   DATA[1506,16] := 1.0;
   DATA[1506,17] := 1.0;
   DATA[1506,18] := 1.0;
   DATA[1506,19] := 2.0;
   DATA[1506,20] := 148.808;
   DATA[1506,21] := 153.5504;
   DATA[1506,22] := 1.711466;
   DATA[1506,23] := 789.4899;
   DATA[1506,24] := 2.0;
   DATA[1506,25] := 2.0;
   DATA[1506,26] := 7.876378;
   DATA[1506,27] := 142.707;
   DATA[1506,28] := 263.1377;
   DATA[1506,29] := 12.11228;
   DATA[1506,30] := 1.723148;
   DATA[1506,31] := 1.297041;
   DATA[1506,32] := 0.7352687;
   DATA[1506,33] := 0.3107325;
   DATA[1506,34] := 2.0;
   DATA[1506,35] := 249.984;
   DATA[1506,36] := 1.665972;
   DATA[1506,37] := 188.7657;
   DATA[1506,38] := 0.000128152;
   DATA[1506,39] := 1.0;
   DATA[1507,1] := 815.2798;
   DATA[1507,2] := 1.0;
   DATA[1507,3] := 1.0;
   DATA[1507,4] := 262.5609;
   DATA[1507,5] := 8.464369;
   DATA[1507,6] := 318.9438;
   DATA[1507,8] := 1.0;
   DATA[1507,9] := 1.0;
   DATA[1507,10] := 1.0;
   DATA[1507,11] := 19.74198;
   DATA[1507,12] := 2.210294;
   DATA[1507,13] := 939.5027;
   DATA[1507,14] := 1.0;
   DATA[1507,15] := 2.0;
   DATA[1507,16] := 1.0;
   DATA[1507,17] := 1.0;
   DATA[1507,18] := 1.0;
   DATA[1507,19] := 2.0;
   DATA[1507,20] := 148.808;
   DATA[1507,21] := 153.5504;
   DATA[1507,22] := 1.711466;
   DATA[1507,23] := 789.5283;
   DATA[1507,24] := 2.0;
   DATA[1507,25] := 2.0;
   DATA[1507,26] := 7.876378;
   DATA[1507,27] := 142.707;
   DATA[1507,28] := 263.0415;
   DATA[1507,29] := 12.11228;
   DATA[1507,30] := 1.723148;
   DATA[1507,31] := 1.290509;
   DATA[1507,32] := 0.7352687;
   DATA[1507,33] := 0.3107325;
   DATA[1507,34] := 2.0;
   DATA[1507,35] := 249.9039;
   DATA[1507,36] := 1.665972;
   DATA[1507,37] := 188.7657;
   DATA[1507,38] := 0.000128152;
   DATA[1507,39] := 1.0;
   DATA[1508,1] := 815.2013;
   DATA[1508,2] := 1.0;
   DATA[1508,3] := 1.0;
   DATA[1508,4] := 262.5609;
   DATA[1508,5] := 8.464369;
   DATA[1508,6] := 318.8413;
   DATA[1508,8] := 1.0;
   DATA[1508,9] := 1.0;
   DATA[1508,10] := 1.0;
   DATA[1508,11] := 19.73878;
   DATA[1508,12] := 2.210934;
   DATA[1508,13] := 939.5428;
   DATA[1508,14] := 1.0;
   DATA[1508,15] := 2.0;
   DATA[1508,16] := 1.0;
   DATA[1508,17] := 1.0;
   DATA[1508,18] := 1.0;
   DATA[1508,19] := 2.0;
   DATA[1508,20] := 148.808;
   DATA[1508,21] := 153.5504;
   DATA[1508,22] := 1.711466;
   DATA[1508,23] := 789.8744;
   DATA[1508,24] := 2.0;
   DATA[1508,25] := 2.0;
   DATA[1508,26] := 7.876378;
   DATA[1508,27] := 142.707;
   DATA[1508,28] := 263.0415;
   DATA[1508,29] := 12.11228;
   DATA[1508,30] := 1.723148;
   DATA[1508,31] := 1.294992;
   DATA[1508,32] := 0.7371892;
   DATA[1508,33] := 0.3107325;
   DATA[1508,34] := 2.0;
   DATA[1508,35] := 249.9039;
   DATA[1508,36] := 1.665972;
   DATA[1508,37] := 188.7657;
   DATA[1508,38] := 0.000128152;
   DATA[1508,39] := 1.0;
   DATA[1509,1] := 814.8873;
   DATA[1509,2] := 1.0;
   DATA[1509,3] := 1.0;
   DATA[1509,4] := 262.5609;
   DATA[1509,5] := 8.464369;
   DATA[1509,6] := 318.6619;
   DATA[1509,8] := 1.0;
   DATA[1509,9] := 1.0;
   DATA[1509,10] := 1.0;
   DATA[1509,11] := 19.75479;
   DATA[1509,12] := 2.211831;
   DATA[1509,13] := 938.982;
   DATA[1509,14] := 1.0;
   DATA[1509,15] := 2.0;
   DATA[1509,16] := 1.0;
   DATA[1509,17] := 1.0;
   DATA[1509,18] := 1.0;
   DATA[1509,19] := 2.0;
   DATA[1509,20] := 148.808;
   DATA[1509,21] := 153.5504;
   DATA[1509,22] := 1.711466;
   DATA[1509,23] := 790.1436;
   DATA[1509,24] := 2.0;
   DATA[1509,25] := 2.0;
   DATA[1509,26] := 7.876378;
   DATA[1509,27] := 142.707;
   DATA[1509,28] := 263.0415;
   DATA[1509,29] := 12.11228;
   DATA[1509,30] := 1.723148;
   DATA[1509,31] := 1.290509;
   DATA[1509,32] := 0.7384694;
   DATA[1509,33] := 0.3107325;
   DATA[1509,34] := 2.0;
   DATA[1509,35] := 249.9039;
   DATA[1509,36] := 1.665972;
   DATA[1509,37] := 188.7657;
   DATA[1509,38] := 0.000128152;
   DATA[1509,39] := 1.0;
   DATA[1510,1] := 814.8088;
   DATA[1510,2] := 1.0;
   DATA[1510,3] := 1.0;
   DATA[1510,4] := 262.5609;
   DATA[1510,5] := 8.464369;
   DATA[1510,6] := 318.6619;
   DATA[1510,8] := 1.0;
   DATA[1510,9] := 1.0;
   DATA[1510,10] := 1.0;
   DATA[1510,11] := 19.7868;
   DATA[1510,12] := 2.211831;
   DATA[1510,13] := 938.7017;
   DATA[1510,14] := 1.0;
   DATA[1510,15] := 2.0;
   DATA[1510,16] := 1.0;
   DATA[1510,17] := 1.0;
   DATA[1510,18] := 1.0;
   DATA[1510,19] := 2.0;
   DATA[1510,20] := 148.808;
   DATA[1510,21] := 153.5504;
   DATA[1510,22] := 1.712748;
   DATA[1510,23] := 789.9513;
   DATA[1510,24] := 2.0;
   DATA[1510,25] := 2.0;
   DATA[1510,26] := 7.876378;
   DATA[1510,27] := 142.707;
   DATA[1510,28] := 263.0415;
   DATA[1510,29] := 12.11228;
   DATA[1510,30] := 1.723148;
   DATA[1510,31] := 1.284104;
   DATA[1510,32] := 0.7384694;
   DATA[1510,33] := 0.3089389;
   DATA[1510,34] := 2.0;
   DATA[1510,35] := 249.9039;
   DATA[1510,36] := 1.665972;
   DATA[1510,37] := 188.8779;
   DATA[1510,38] := 0.000128152;
   DATA[1510,39] := 1.0;
   DATA[1511,1] := 815.2798;
   DATA[1511,2] := 1.0;
   DATA[1511,3] := 1.0;
   DATA[1511,4] := 262.5609;
   DATA[1511,5] := 8.462446;
   DATA[1511,6] := 318.6619;
   DATA[1511,8] := 1.0;
   DATA[1511,9] := 1.0;
   DATA[1511,10] := 1.0;
   DATA[1511,11] := 19.69396;
   DATA[1511,12] := 2.209397;
   DATA[1511,13] := 937.9406;
   DATA[1511,14] := 1.0;
   DATA[1511,15] := 2.0;
   DATA[1511,16] := 1.0;
   DATA[1511,17] := 1.0;
   DATA[1511,18] := 1.0;
   DATA[1511,19] := 2.0;
   DATA[1511,20] := 148.808;
   DATA[1511,21] := 153.5504;
   DATA[1511,22] := 1.712748;
   DATA[1511,23] := 789.7975;
   DATA[1511,24] := 2.0;
   DATA[1511,25] := 2.0;
   DATA[1511,26] := 7.876378;
   DATA[1511,27] := 142.707;
   DATA[1511,28] := 263.0415;
   DATA[1511,29] := 12.11228;
   DATA[1511,30] := 1.723148;
   DATA[1511,31] := 1.287947;
   DATA[1511,32] := 0.7384694;
   DATA[1511,33] := 0.3089389;
   DATA[1511,34] := 2.0;
   DATA[1511,35] := 249.9039;
   DATA[1511,36] := 1.665972;
   DATA[1511,37] := 188.8779;
   DATA[1511,38] := 0.000128152;
   DATA[1511,39] := 1.0;
   DATA[1512,1] := 815.005;
   DATA[1512,2] := 1.0;
   DATA[1512,3] := 1.0;
   DATA[1512,4] := 262.5609;
   DATA[1512,5] := 8.462446;
   DATA[1512,6] := 318.6619;
   DATA[1512,8] := 1.0;
   DATA[1512,9] := 1.0;
   DATA[1512,10] := 1.0;
   DATA[1512,11] := 19.69076;
   DATA[1512,12] := 2.209397;
   DATA[1512,13] := 937.5401;
   DATA[1512,14] := 1.0;
   DATA[1512,15] := 2.0;
   DATA[1512,16] := 1.0;
   DATA[1512,17] := 1.0;
   DATA[1512,18] := 1.0;
   DATA[1512,19] := 2.0;
   DATA[1512,20] := 148.808;
   DATA[1512,21] := 153.5504;
   DATA[1512,22] := 1.712748;
   DATA[1512,23] := 790.1051;
   DATA[1512,24] := 2.0;
   DATA[1512,25] := 2.0;
   DATA[1512,26] := 7.876378;
   DATA[1512,27] := 142.707;
   DATA[1512,28] := 263.0415;
   DATA[1512,29] := 12.11228;
   DATA[1512,30] := 1.723148;
   DATA[1512,31] := 1.285641;
   DATA[1512,32] := 0.7384694;
   DATA[1512,33] := 0.3083624;
   DATA[1512,34] := 2.0;
   DATA[1512,35] := 250.0;
   DATA[1512,36] := 1.665972;
   DATA[1512,37] := 188.8779;
   DATA[1512,38] := 0.000128152;
   DATA[1512,39] := 1.0;
   DATA[1513,1] := 815.4761;
   DATA[1513,2] := 1.0;
   DATA[1513,3] := 1.0;
   DATA[1513,4] := 262.5609;
   DATA[1513,5] := 8.462446;
   DATA[1513,6] := 318.6619;
   DATA[1513,8] := 1.0;
   DATA[1513,9] := 1.0;
   DATA[1513,10] := 1.0;
   DATA[1513,11] := 19.67155;
   DATA[1513,12] := 2.209397;
   DATA[1513,13] := 936.8992;
   DATA[1513,14] := 1.0;
   DATA[1513,15] := 2.0;
   DATA[1513,16] := 1.0;
   DATA[1513,17] := 1.0;
   DATA[1513,18] := 1.0;
   DATA[1513,19] := 2.0;
   DATA[1513,20] := 148.808;
   DATA[1513,21] := 153.6273;
   DATA[1513,22] := 1.712748;
   DATA[1513,23] := 789.9128;
   DATA[1513,24] := 2.0;
   DATA[1513,25] := 2.0;
   DATA[1513,26] := 7.876378;
   DATA[1513,27] := 142.707;
   DATA[1513,28] := 263.0095;
   DATA[1513,29] := 12.11228;
   DATA[1513,30] := 1.723148;
   DATA[1513,31] := 1.288075;
   DATA[1513,32] := 0.7384694;
   DATA[1513,33] := 0.3082983;
   DATA[1513,34] := 2.0;
   DATA[1513,35] := 250.016;
   DATA[1513,36] := 1.665972;
   DATA[1513,37] := 188.8779;
   DATA[1513,38] := 0.000128152;
   DATA[1513,39] := 1.0;
   DATA[1514,1] := 815.4761;
   DATA[1514,2] := 1.0;
   DATA[1514,3] := 1.0;
   DATA[1514,4] := 262.5609;
   DATA[1514,5] := 8.462446;
   DATA[1514,6] := 318.8413;
   DATA[1514,8] := 1.0;
   DATA[1514,9] := 1.0;
   DATA[1514,10] := 1.0;
   DATA[1514,11] := 19.65235;
   DATA[1514,12] := 2.209397;
   DATA[1514,13] := 936.8591;
   DATA[1514,14] := 1.0;
   DATA[1514,15] := 2.0;
   DATA[1514,16] := 1.0;
   DATA[1514,17] := 1.0;
   DATA[1514,18] := 1.0;
   DATA[1514,19] := 2.0;
   DATA[1514,20] := 148.808;
   DATA[1514,21] := 153.6273;
   DATA[1514,22] := 1.712876;
   DATA[1514,23] := 790.3358;
   DATA[1514,24] := 2.0;
   DATA[1514,25] := 2.0;
   DATA[1514,26] := 7.876378;
   DATA[1514,27] := 142.707;
   DATA[1514,28] := 262.9454;
   DATA[1514,29] := 12.11228;
   DATA[1514,30] := 1.723148;
   DATA[1514,31] := 1.28167;
   DATA[1514,32] := 0.7384694;
   DATA[1514,33] := 0.3082983;
   DATA[1514,34] := 2.0;
   DATA[1514,35] := 250.016;
   DATA[1514,36] := 1.665972;
   DATA[1514,37] := 188.8779;
   DATA[1514,38] := 0.000128152;
   DATA[1514,39] := 1.0;
   DATA[1515,1] := 815.4761;
   DATA[1515,2] := 1.0;
   DATA[1515,3] := 1.0;
   DATA[1515,4] := 262.5609;
   DATA[1515,5] := 8.462446;
   DATA[1515,6] := 318.8413;
   DATA[1515,8] := 1.0;
   DATA[1515,9] := 1.0;
   DATA[1515,10] := 1.0;
   DATA[1515,11] := 19.65235;
   DATA[1515,12] := 2.209397;
   DATA[1515,13] := 936.4586;
   DATA[1515,14] := 1.0;
   DATA[1515,15] := 2.0;
   DATA[1515,16] := 1.0;
   DATA[1515,17] := 1.0;
   DATA[1515,18] := 1.0;
   DATA[1515,19] := 2.0;
   DATA[1515,20] := 148.808;
   DATA[1515,21] := 153.858;
   DATA[1515,22] := 1.712876;
   DATA[1515,23] := 790.5281;
   DATA[1515,24] := 2.0;
   DATA[1515,25] := 2.0;
   DATA[1515,26] := 7.876378;
   DATA[1515,27] := 142.707;
   DATA[1515,28] := 262.9454;
   DATA[1515,29] := 12.11228;
   DATA[1515,30] := 1.721866;
   DATA[1515,31] := 1.286922;
   DATA[1515,32] := 0.7384694;
   DATA[1515,33] := 0.3082983;
   DATA[1515,34] := 2.0;
   DATA[1515,35] := 250.016;
   DATA[1515,36] := 1.665972;
   DATA[1515,37] := 188.8779;
   DATA[1515,38] := 0.000128152;
   DATA[1515,39] := 1.0;
   DATA[1516,1] := 815.1228;
   DATA[1516,2] := 1.0;
   DATA[1516,3] := 1.0;
   DATA[1516,4] := 262.5609;
   DATA[1516,5] := 8.462446;
   DATA[1516,6] := 318.8413;
   DATA[1516,8] := 1.0;
   DATA[1516,9] := 1.0;
   DATA[1516,10] := 1.0;
   DATA[1516,11] := 19.73558;
   DATA[1516,12] := 2.209397;
   DATA[1516,13] := 935.8979;
   DATA[1516,14] := 1.0;
   DATA[1516,15] := 2.0;
   DATA[1516,16] := 1.0;
   DATA[1516,17] := 1.0;
   DATA[1516,18] := 1.0;
   DATA[1516,19] := 2.0;
   DATA[1516,20] := 148.808;
   DATA[1516,21] := 153.858;
   DATA[1516,22] := 1.711595;
   DATA[1516,23] := 790.6819;
   DATA[1516,24] := 2.0;
   DATA[1516,25] := 2.0;
   DATA[1516,26] := 7.876378;
   DATA[1516,27] := 142.707;
   DATA[1516,28] := 262.9454;
   DATA[1516,29] := 12.11228;
   DATA[1516,30] := 1.721866;
   DATA[1516,31] := 1.288203;
   DATA[1516,32] := 0.7384694;
   DATA[1516,33] := 0.3082983;
   DATA[1516,34] := 2.0;
   DATA[1516,35] := 250.016;
   DATA[1516,36] := 1.665972;
   DATA[1516,37] := 188.8779;
   DATA[1516,38] := 0.000128152;
   DATA[1516,39] := 1.0;
   DATA[1517,1] := 814.8873;
   DATA[1517,2] := 1.0;
   DATA[1517,3] := 1.0;
   DATA[1517,4] := 262.5609;
   DATA[1517,5] := 8.462446;
   DATA[1517,6] := 318.8413;
   DATA[1517,8] := 1.0;
   DATA[1517,9] := 1.0;
   DATA[1517,10] := 1.0;
   DATA[1517,11] := 19.77079;
   DATA[1517,12] := 2.211318;
   DATA[1517,13] := 935.8578;
   DATA[1517,14] := 1.0;
   DATA[1517,15] := 2.0;
   DATA[1517,16] := 1.0;
   DATA[1517,17] := 1.0;
   DATA[1517,18] := 1.0;
   DATA[1517,19] := 2.0;
   DATA[1517,20] := 148.808;
   DATA[1517,21] := 153.858;
   DATA[1517,22] := 1.710185;
   DATA[1517,23] := 790.6434;
   DATA[1517,24] := 2.0;
   DATA[1517,25] := 2.0;
   DATA[1517,26] := 7.876378;
   DATA[1517,27] := 142.707;
   DATA[1517,28] := 262.9454;
   DATA[1517,29] := 12.11228;
   DATA[1517,30] := 1.723148;
   DATA[1517,31] := 1.281798;
   DATA[1517,32] := 0.7374452;
   DATA[1517,33] := 0.3082983;
   DATA[1517,34] := 2.0;
   DATA[1517,35] := 250.016;
   DATA[1517,36] := 1.665972;
   DATA[1517,37] := 188.8779;
   DATA[1517,38] := 0.000128152;
   DATA[1517,39] := 1.0;
   DATA[1518,1] := 815.2013;
   DATA[1518,2] := 1.0;
   DATA[1518,3] := 1.0;
   DATA[1518,4] := 262.5609;
   DATA[1518,5] := 8.462446;
   DATA[1518,6] := 318.8413;
   DATA[1518,8] := 1.0;
   DATA[1518,9] := 1.0;
   DATA[1518,10] := 1.0;
   DATA[1518,11] := 19.8028;
   DATA[1518,12] := 2.211575;
   DATA[1518,13] := 934.8965;
   DATA[1518,14] := 1.0;
   DATA[1518,15] := 2.0;
   DATA[1518,16] := 1.0;
   DATA[1518,17] := 1.0;
   DATA[1518,18] := 1.0;
   DATA[1518,19] := 2.0;
   DATA[1518,20] := 148.808;
   DATA[1518,21] := 153.7298;
   DATA[1518,22] := 1.710185;
   DATA[1518,23] := 790.5281;
   DATA[1518,24] := 2.0;
   DATA[1518,25] := 2.0;
   DATA[1518,26] := 7.876378;
   DATA[1518,27] := 142.707;
   DATA[1518,28] := 262.9454;
   DATA[1518,29] := 12.11228;
   DATA[1518,30] := 1.724045;
   DATA[1518,31] := 1.281798;
   DATA[1518,32] := 0.7374452;
   DATA[1518,33] := 0.3082983;
   DATA[1518,34] := 2.0;
   DATA[1518,35] := 250.016;
   DATA[1518,36] := 1.665972;
   DATA[1518,37] := 188.8779;
   DATA[1518,38] := 0.000128152;
   DATA[1518,39] := 1.0;
   DATA[1519,1] := 815.0835;
   DATA[1519,2] := 1.0;
   DATA[1519,3] := 1.0;
   DATA[1519,4] := 262.5609;
   DATA[1519,5] := 8.462446;
   DATA[1519,6] := 318.8413;
   DATA[1519,8] := 1.0;
   DATA[1519,9] := 1.0;
   DATA[1519,10] := 1.0;
   DATA[1519,11] := 19.83162;
   DATA[1519,12] := 2.211575;
   DATA[1519,13] := 933.9753;
   DATA[1519,14] := 1.0;
   DATA[1519,15] := 2.0;
   DATA[1519,16] := 1.0;
   DATA[1519,17] := 1.0;
   DATA[1519,18] := 1.0;
   DATA[1519,19] := 2.0;
   DATA[1519,20] := 148.808;
   DATA[1519,21] := 153.7298;
   DATA[1519,22] := 1.710185;
   DATA[1519,23] := 790.2589;
   DATA[1519,24] := 2.0;
   DATA[1519,25] := 2.0;
   DATA[1519,26] := 7.876378;
   DATA[1519,27] := 142.707;
   DATA[1519,28] := 262.9454;
   DATA[1519,29] := 12.11228;
   DATA[1519,30] := 1.724045;
   DATA[1519,31] := 1.288587;
   DATA[1519,32] := 0.7374452;
   DATA[1519,33] := 0.3082983;
   DATA[1519,34] := 2.0;
   DATA[1519,35] := 250.016;
   DATA[1519,36] := 1.665972;
   DATA[1519,37] := 188.7977;
   DATA[1519,38] := 0.000128152;
   DATA[1519,39] := 1.0;
   DATA[1520,1] := 815.0835;
   DATA[1520,2] := 1.0;
   DATA[1520,3] := 1.0;
   DATA[1520,4] := 262.5609;
   DATA[1520,5] := 8.462446;
   DATA[1520,6] := 318.8413;
   DATA[1520,8] := 1.0;
   DATA[1520,9] := 1.0;
   DATA[1520,10] := 1.0;
   DATA[1520,11] := 19.83162;
   DATA[1520,12] := 2.211575;
   DATA[1520,13] := 933.9753;
   DATA[1520,14] := 1.0;
   DATA[1520,15] := 2.0;
   DATA[1520,16] := 1.0;
   DATA[1520,17] := 1.0;
   DATA[1520,18] := 1.0;
   DATA[1520,19] := 2.0;
   DATA[1520,20] := 148.808;
   DATA[1520,21] := 153.7298;
   DATA[1520,22] := 1.710185;
   DATA[1520,23] := 790.0667;
   DATA[1520,24] := 2.0;
   DATA[1520,25] := 2.0;
   DATA[1520,26] := 7.876378;
   DATA[1520,27] := 142.707;
   DATA[1520,28] := 262.9454;
   DATA[1520,29] := 12.11228;
   DATA[1520,30] := 1.724045;
   DATA[1520,31] := 1.291277;
   DATA[1520,32] := 0.7359089;
   DATA[1520,33] := 0.3082983;
   DATA[1520,34] := 2.0;
   DATA[1520,35] := 250.016;
   DATA[1520,36] := 1.665972;
   DATA[1520,37] := 188.7977;
   DATA[1520,38] := 0.000128152;
   DATA[1520,39] := 1.0;
   DATA[1521,1] := 815.005;
   DATA[1521,2] := 1.0;
   DATA[1521,3] := 1.0;
   DATA[1521,4] := 262.5609;
   DATA[1521,5] := 8.462446;
   DATA[1521,6] := 318.8413;
   DATA[1521,8] := 1.0;
   DATA[1521,9] := 1.0;
   DATA[1521,10] := 1.0;
   DATA[1521,11] := 19.83162;
   DATA[1521,12] := 2.214265;
   DATA[1521,13] := 933.775;
   DATA[1521,14] := 1.0;
   DATA[1521,15] := 2.0;
   DATA[1521,16] := 1.0;
   DATA[1521,17] := 1.0;
   DATA[1521,18] := 1.0;
   DATA[1521,19] := 2.0;
   DATA[1521,20] := 148.808;
   DATA[1521,21] := 153.7298;
   DATA[1521,22] := 1.711723;
   DATA[1521,23] := 789.8744;
   DATA[1521,24] := 2.0;
   DATA[1521,25] := 2.0;
   DATA[1521,26] := 7.876378;
   DATA[1521,27] := 142.707;
   DATA[1521,28] := 262.9454;
   DATA[1521,29] := 12.11228;
   DATA[1521,30] := 1.724045;
   DATA[1521,31] := 1.30178;
   DATA[1521,32] := 0.7359089;
   DATA[1521,33] := 0.3082983;
   DATA[1521,34] := 2.0;
   DATA[1521,35] := 250.016;
   DATA[1521,36] := 1.665972;
   DATA[1521,37] := 188.7977;
   DATA[1521,38] := 0.000128152;
   DATA[1521,39] := 1.0;
   DATA[1522,1] := 815.2013;
   DATA[1522,2] := 1.0;
   DATA[1522,3] := 1.0;
   DATA[1522,4] := 262.5609;
   DATA[1522,5] := 8.463728;
   DATA[1522,6] := 318.8413;
   DATA[1522,8] := 1.0;
   DATA[1522,9] := 1.0;
   DATA[1522,10] := 1.0;
   DATA[1522,11] := 19.77399;
   DATA[1522,12] := 2.214265;
   DATA[1522,13] := 933.3745;
   DATA[1522,14] := 1.0;
   DATA[1522,15] := 2.0;
   DATA[1522,16] := 1.0;
   DATA[1522,17] := 1.0;
   DATA[1522,18] := 1.0;
   DATA[1522,19] := 2.0;
   DATA[1522,20] := 148.808;
   DATA[1522,21] := 153.7298;
   DATA[1522,22] := 1.713389;
   DATA[1522,23] := 789.6052;
   DATA[1522,24] := 2.0;
   DATA[1522,25] := 2.0;
   DATA[1522,26] := 7.876378;
   DATA[1522,27] := 142.707;
   DATA[1522,28] := 262.9454;
   DATA[1522,29] := 12.11228;
   DATA[1522,30] := 1.724045;
   DATA[1522,31] := 1.29576;
   DATA[1522,32] := 0.7359089;
   DATA[1522,33] := 0.3082983;
   DATA[1522,34] := 2.0;
   DATA[1522,35] := 250.016;
   DATA[1522,36] := 1.665972;
   DATA[1522,37] := 188.7977;
   DATA[1522,38] := 0.000128152;
   DATA[1522,39] := 1.0;
   DATA[1523,1] := 815.162;
   DATA[1523,2] := 1.0;
   DATA[1523,3] := 1.0;
   DATA[1523,4] := 262.5609;
   DATA[1523,5] := 8.46501;
   DATA[1523,6] := 318.8413;
   DATA[1523,8] := 1.0;
   DATA[1523,9] := 1.0;
   DATA[1523,10] := 1.0;
   DATA[1523,11] := 19.77079;
   DATA[1523,12] := 2.214265;
   DATA[1523,13] := 933.0941;
   DATA[1523,14] := 1.0;
   DATA[1523,15] := 2.0;
   DATA[1523,16] := 1.0;
   DATA[1523,17] := 1.0;
   DATA[1523,18] := 1.0;
   DATA[1523,19] := 2.0;
   DATA[1523,20] := 148.808;
   DATA[1523,21] := 153.7298;
   DATA[1523,22] := 1.713389;
   DATA[1523,23] := 789.9513;
   DATA[1523,24] := 2.0;
   DATA[1523,25] := 2.0;
   DATA[1523,26] := 7.876378;
   DATA[1523,27] := 142.707;
   DATA[1523,28] := 262.9454;
   DATA[1523,29] := 12.11228;
   DATA[1523,30] := 1.721738;
   DATA[1523,31] := 1.275906;
   DATA[1523,32] := 0.7359089;
   DATA[1523,33] := 0.3082983;
   DATA[1523,34] := 2.0;
   DATA[1523,35] := 250.016;
   DATA[1523,36] := 1.665972;
   DATA[1523,37] := 188.7977;
   DATA[1523,38] := 0.000128152;
   DATA[1523,39] := 1.0;
   DATA[1524,1] := 815.3583;
   DATA[1524,2] := 1.0;
   DATA[1524,3] := 1.0;
   DATA[1524,4] := 262.5609;
   DATA[1524,5] := 8.46501;
   DATA[1524,6] := 318.8413;
   DATA[1524,8] := 1.0;
   DATA[1524,9] := 1.0;
   DATA[1524,10] := 1.0;
   DATA[1524,11] := 19.74838;
   DATA[1524,12] := 2.214137;
   DATA[1524,13] := 932.5734;
   DATA[1524,14] := 1.0;
   DATA[1524,15] := 2.0;
   DATA[1524,16] := 1.0;
   DATA[1524,17] := 1.0;
   DATA[1524,18] := 1.0;
   DATA[1524,19] := 2.0;
   DATA[1524,20] := 148.808;
   DATA[1524,21] := 153.7298;
   DATA[1524,22] := 1.713389;
   DATA[1524,23] := 789.8744;
   DATA[1524,24] := 2.0;
   DATA[1524,25] := 2.0;
   DATA[1524,26] := 7.876378;
   DATA[1524,27] := 142.707;
   DATA[1524,28] := 262.9454;
   DATA[1524,29] := 12.11228;
   DATA[1524,30] := 1.720969;
   DATA[1524,31] := 1.271551;
   DATA[1524,32] := 0.7351407;
   DATA[1524,33] := 0.3082983;
   DATA[1524,34] := 2.0;
   DATA[1524,35] := 250.016;
   DATA[1524,36] := 1.665972;
   DATA[1524,37] := 188.7977;
   DATA[1524,38] := 0.000128152;
   DATA[1524,39] := 1.0;
   DATA[1525,1] := 815.162;
   DATA[1525,2] := 1.0;
   DATA[1525,3] := 1.0;
   DATA[1525,4] := 262.5609;
   DATA[1525,5] := 8.46501;
   DATA[1525,6] := 318.8413;
   DATA[1525,8] := 1.0;
   DATA[1525,9] := 1.0;
   DATA[1525,10] := 1.0;
   DATA[1525,11] := 19.74838;
   DATA[1525,12] := 2.212215;
   DATA[1525,13] := 932.4933;
   DATA[1525,14] := 1.0;
   DATA[1525,15] := 2.0;
   DATA[1525,16] := 1.0;
   DATA[1525,17] := 1.0;
   DATA[1525,18] := 1.0;
   DATA[1525,19] := 2.0;
   DATA[1525,20] := 148.808;
   DATA[1525,21] := 153.7298;
   DATA[1525,22] := 1.711082;
   DATA[1525,23] := 789.9513;
   DATA[1525,24] := 2.0;
   DATA[1525,25] := 2.0;
   DATA[1525,26] := 7.876378;
   DATA[1525,27] := 142.707;
   DATA[1525,28] := 262.9454;
   DATA[1525,29] := 12.11228;
   DATA[1525,30] := 1.719559;
   DATA[1525,31] := 1.271551;
   DATA[1525,32] := 0.7348846;
   DATA[1525,33] := 0.3082983;
   DATA[1525,34] := 2.0;
   DATA[1525,35] := 250.016;
   DATA[1525,36] := 1.665972;
   DATA[1525,37] := 188.7977;
   DATA[1525,38] := 0.000128152;
   DATA[1525,39] := 1.0;
   DATA[1526,1] := 815.2013;
   DATA[1526,2] := 1.0;
   DATA[1526,3] := 1.0;
   DATA[1526,4] := 262.5609;
   DATA[1526,5] := 8.46501;
   DATA[1526,6] := 318.8413;
   DATA[1526,8] := 1.0;
   DATA[1526,9] := 1.0;
   DATA[1526,10] := 1.0;
   DATA[1526,11] := 19.71637;
   DATA[1526,12] := 2.212215;
   DATA[1526,13] := 931.7723;
   DATA[1526,14] := 1.0;
   DATA[1526,15] := 2.0;
   DATA[1526,16] := 1.0;
   DATA[1526,17] := 1.0;
   DATA[1526,18] := 1.0;
   DATA[1526,19] := 2.0;
   DATA[1526,20] := 148.808;
   DATA[1526,21] := 153.7298;
   DATA[1526,22] := 1.711082;
   DATA[1526,23] := 789.759;
   DATA[1526,24] := 2.0;
   DATA[1526,25] := 2.0;
   DATA[1526,26] := 7.876378;
   DATA[1526,27] := 142.707;
   DATA[1526,28] := 262.9454;
   DATA[1526,29] := 12.11228;
   DATA[1526,30] := 1.719559;
   DATA[1526,31] := 1.285001;
   DATA[1526,32] := 0.7348846;
   DATA[1526,33] := 0.3082983;
   DATA[1526,34] := 2.0;
   DATA[1526,35] := 250.016;
   DATA[1526,36] := 1.665972;
   DATA[1526,37] := 188.7977;
   DATA[1526,38] := 0.000128152;
   DATA[1526,39] := 1.0;
   DATA[1527,1] := 815.319;
   DATA[1527,2] := 1.0;
   DATA[1527,3] := 1.0;
   DATA[1527,4] := 262.5609;
   DATA[1527,5] := 8.46501;
   DATA[1527,6] := 318.8413;
   DATA[1527,8] := 1.0;
   DATA[1527,9] := 1.0;
   DATA[1527,10] := 1.0;
   DATA[1527,11] := 19.65875;
   DATA[1527,12] := 2.21055;
   DATA[1527,13] := 931.532;
   DATA[1527,14] := 1.0;
   DATA[1527,15] := 2.0;
   DATA[1527,16] := 1.0;
   DATA[1527,17] := 1.0;
   DATA[1527,18] := 1.0;
   DATA[1527,19] := 2.0;
   DATA[1527,20] := 148.808;
   DATA[1527,21] := 153.7298;
   DATA[1527,22] := 1.711082;
   DATA[1527,23] := 789.9128;
   DATA[1527,24] := 2.0;
   DATA[1527,25] := 2.0;
   DATA[1527,26] := 7.876378;
   DATA[1527,27] := 142.707;
   DATA[1527,28] := 262.9454;
   DATA[1527,29] := 12.11228;
   DATA[1527,30] := 1.719559;
   DATA[1527,31] := 1.290893;
   DATA[1527,32] := 0.7348846;
   DATA[1527,33] := 0.3082983;
   DATA[1527,34] := 2.0;
   DATA[1527,35] := 250.016;
   DATA[1527,36] := 1.746067;
   DATA[1527,37] := 188.8618;
   DATA[1527,38] := 0.000128152;
   DATA[1527,39] := 1.0;
   DATA[1528,1] := 815.2013;
   DATA[1528,2] := 1.0;
   DATA[1528,3] := 1.0;
   DATA[1528,4] := 262.5609;
   DATA[1528,5] := 8.46501;
   DATA[1528,6] := 318.8413;
   DATA[1528,8] := 1.0;
   DATA[1528,9] := 1.0;
   DATA[1528,10] := 1.0;
   DATA[1528,11] := 19.62033;
   DATA[1528,12] := 2.210294;
   DATA[1528,13] := 930.9713;
   DATA[1528,14] := 1.0;
   DATA[1528,15] := 2.0;
   DATA[1528,16] := 1.0;
   DATA[1528,17] := 1.0;
   DATA[1528,18] := 1.0;
   DATA[1528,19] := 2.0;
   DATA[1528,20] := 148.808;
   DATA[1528,21] := 153.7298;
   DATA[1528,22] := 1.711082;
   DATA[1528,23] := 789.9128;
   DATA[1528,24] := 2.0;
   DATA[1528,25] := 2.0;
   DATA[1528,26] := 7.876378;
   DATA[1528,27] := 142.5788;
   DATA[1528,28] := 262.9454;
   DATA[1528,29] := 12.11228;
   DATA[1528,30] := 1.719559;
   DATA[1528,31] := 1.291405;
   DATA[1528,32] := 0.7348846;
   DATA[1528,33] := 0.3082983;
   DATA[1528,34] := 2.0;
   DATA[1528,35] := 250.016;
   DATA[1528,36] := 1.746067;
   DATA[1528,37] := 188.8618;
   DATA[1528,38] := 0.000128152;
   DATA[1528,39] := 1.0;
   DATA[1529,1] := 815.1228;
   DATA[1529,2] := 1.0;
   DATA[1529,3] := 1.0;
   DATA[1529,4] := 262.5609;
   DATA[1529,5] := 8.46501;
   DATA[1529,6] := 318.8413;
   DATA[1529,8] := 1.0;
   DATA[1529,9] := 1.0;
   DATA[1529,10] := 1.0;
   DATA[1529,11] := 19.62033;
   DATA[1529,12] := 2.210294;
   DATA[1529,13] := 930.6508;
   DATA[1529,14] := 1.0;
   DATA[1529,15] := 2.0;
   DATA[1529,16] := 1.0;
   DATA[1529,17] := 1.0;
   DATA[1529,18] := 1.0;
   DATA[1529,19] := 2.0;
   DATA[1529,20] := 148.808;
   DATA[1529,21] := 153.7298;
   DATA[1529,22] := 1.711979;
   DATA[1529,23] := 789.9897;
   DATA[1529,24] := 2.0;
   DATA[1529,25] := 2.0;
   DATA[1529,26] := 7.876378;
   DATA[1529,27] := 142.5788;
   DATA[1529,28] := 262.9454;
   DATA[1529,29] := 12.11228;
   DATA[1529,30] := 1.719559;
   DATA[1529,31] := 1.291405;
   DATA[1529,32] := 0.7348846;
   DATA[1529,33] := 0.3082983;
   DATA[1529,34] := 2.0;
   DATA[1529,35] := 250.016;
   DATA[1529,36] := 1.746067;
   DATA[1529,37] := 188.8618;
   DATA[1529,38] := 0.000128152;
   DATA[1529,39] := 1.0;
   DATA[1530,1] := 815.1228;
   DATA[1530,2] := 1.0;
   DATA[1530,3] := 1.0;
   DATA[1530,4] := 262.5609;
   DATA[1530,5] := 8.46501;
   DATA[1530,6] := 318.8413;
   DATA[1530,8] := 1.0;
   DATA[1530,9] := 1.0;
   DATA[1530,10] := 1.0;
   DATA[1530,11] := 19.68756;
   DATA[1530,12] := 2.210294;
   DATA[1530,13] := 930.5306;
   DATA[1530,14] := 1.0;
   DATA[1530,15] := 2.0;
   DATA[1530,16] := 1.0;
   DATA[1530,17] := 1.0;
   DATA[1530,18] := 1.0;
   DATA[1530,19] := 2.0;
   DATA[1530,20] := 148.808;
   DATA[1530,21] := 153.7298;
   DATA[1530,22] := 1.714542;
   DATA[1530,23] := 789.7975;
   DATA[1530,24] := 2.0;
   DATA[1530,25] := 2.0;
   DATA[1530,26] := 7.876378;
   DATA[1530,27] := 142.5788;
   DATA[1530,28] := 262.9454;
   DATA[1530,29] := 12.11228;
   DATA[1530,30] := 1.719559;
   DATA[1530,31] := 1.28436;
   DATA[1530,32] := 0.7348846;
   DATA[1530,33] := 0.3082983;
   DATA[1530,34] := 2.0;
   DATA[1530,35] := 250.1602;
   DATA[1530,36] := 1.521802;
   DATA[1530,37] := 188.9259;
   DATA[1530,38] := 0.000128152;
   DATA[1530,39] := 1.0;
   DATA[1531,1] := 815.1228;
   DATA[1531,2] := 1.0;
   DATA[1531,3] := 1.0;
   DATA[1531,4] := 262.5609;
   DATA[1531,5] := 8.46501;
   DATA[1531,6] := 318.8413;
   DATA[1531,8] := 1.0;
   DATA[1531,9] := 1.0;
   DATA[1531,10] := 1.0;
   DATA[1531,11] := 19.72598;
   DATA[1531,12] := 2.211831;
   DATA[1531,13] := 930.05;
   DATA[1531,14] := 1.0;
   DATA[1531,15] := 2.0;
   DATA[1531,16] := 1.0;
   DATA[1531,17] := 1.0;
   DATA[1531,18] := 1.0;
   DATA[1531,19] := 2.0;
   DATA[1531,20] := 148.808;
   DATA[1531,21] := 153.7298;
   DATA[1531,22] := 1.714926;
   DATA[1531,23] := 789.759;
   DATA[1531,24] := 2.0;
   DATA[1531,25] := 2.0;
   DATA[1531,26] := 7.876378;
   DATA[1531,27] := 142.5788;
   DATA[1531,28] := 262.9454;
   DATA[1531,29] := 12.11228;
   DATA[1531,30] := 1.720969;
   DATA[1531,31] := 1.290893;
   DATA[1531,32] := 0.7348846;
   DATA[1531,33] := 0.3082983;
   DATA[1531,34] := 2.0;
   DATA[1531,35] := 250.1602;
   DATA[1531,36] := 1.521802;
   DATA[1531,37] := 189.022;
   DATA[1531,38] := 0.000128152;
   DATA[1531,39] := 1.0;
   DATA[1532,1] := 815.1228;
   DATA[1532,2] := 1.0;
   DATA[1532,3] := 1.0;
   DATA[1532,4] := 262.5609;
   DATA[1532,5] := 8.46501;
   DATA[1532,6] := 318.8413;
   DATA[1532,8] := 1.0;
   DATA[1532,9] := 1.0;
   DATA[1532,10] := 1.0;
   DATA[1532,11] := 19.73558;
   DATA[1532,12] := 2.212728;
   DATA[1532,13] := 929.249;
   DATA[1532,14] := 1.0;
   DATA[1532,15] := 2.0;
   DATA[1532,16] := 1.0;
   DATA[1532,17] := 1.0;
   DATA[1532,18] := 1.0;
   DATA[1532,19] := 2.0;
   DATA[1532,20] := 148.808;
   DATA[1532,21] := 153.7298;
   DATA[1532,22] := 1.717361;
   DATA[1532,23] := 790.2589;
   DATA[1532,24] := 2.0;
   DATA[1532,25] := 2.0;
   DATA[1532,26] := 7.876378;
   DATA[1532,27] := 142.5788;
   DATA[1532,28] := 262.9454;
   DATA[1532,29] := 12.11228;
   DATA[1532,30] := 1.724686;
   DATA[1532,31] := 1.30178;
   DATA[1532,32] := 0.7348846;
   DATA[1532,33] := 0.3082983;
   DATA[1532,34] := 2.0;
   DATA[1532,35] := 250.3365;
   DATA[1532,36] := 1.649953;
   DATA[1532,37] := 189.022;
   DATA[1532,38] := 0.000128152;
   DATA[1532,39] := 1.0;
   DATA[1533,1] := 815.005;
   DATA[1533,2] := 1.0;
   DATA[1533,3] := 1.0;
   DATA[1533,4] := 262.5609;
   DATA[1533,5] := 8.46501;
   DATA[1533,6] := 318.8413;
   DATA[1533,8] := 1.0;
   DATA[1533,9] := 1.0;
   DATA[1533,10] := 1.0;
   DATA[1533,11] := 19.73558;
   DATA[1533,12] := 2.213881;
   DATA[1533,13] := 928.528;
   DATA[1533,14] := 1.0;
   DATA[1533,15] := 2.0;
   DATA[1533,16] := 1.0;
   DATA[1533,17] := 1.0;
   DATA[1533,18] := 1.0;
   DATA[1533,19] := 2.0;
   DATA[1533,20] := 148.808;
   DATA[1533,21] := 153.858;
   DATA[1533,22] := 1.717874;
   DATA[1533,23] := 790.5665;
   DATA[1533,24] := 2.0;
   DATA[1533,25] := 2.0;
   DATA[1533,26] := 7.876378;
   DATA[1533,27] := 142.5788;
   DATA[1533,28] := 262.9454;
   DATA[1533,29] := 12.11228;
   DATA[1533,30] := 1.724686;
   DATA[1533,31] := 1.30178;
   DATA[1533,32] := 0.7348846;
   DATA[1533,33] := 0.3082983;
   DATA[1533,34] := 2.0;
   DATA[1533,35] := 250.3365;
   DATA[1533,36] := 1.649953;
   DATA[1533,37] := 189.0541;
   DATA[1533,38] := 0.000128152;
   DATA[1533,39] := 1.0;
   DATA[1534,1] := 814.7695;
   DATA[1534,2] := 1.0;
   DATA[1534,3] := 1.0;
   DATA[1534,4] := 262.6891;
   DATA[1534,5] := 8.46501;
   DATA[1534,6] := 318.8413;
   DATA[1534,8] := 1.0;
   DATA[1534,9] := 1.0;
   DATA[1534,10] := 1.0;
   DATA[1534,11] := 19.75159;
   DATA[1534,12] := 2.213881;
   DATA[1534,13] := 928.0073;
   DATA[1534,14] := 1.0;
   DATA[1534,15] := 2.0;
   DATA[1534,16] := 1.0;
   DATA[1534,17] := 1.0;
   DATA[1534,18] := 1.0;
   DATA[1534,19] := 2.0;
   DATA[1534,20] := 148.808;
   DATA[1534,21] := 153.858;
   DATA[1534,22] := 1.717874;
   DATA[1534,23] := 790.9126;
   DATA[1534,24] := 2.0;
   DATA[1534,25] := 2.0;
   DATA[1534,26] := 7.876378;
   DATA[1534,27] := 142.5788;
   DATA[1534,28] := 262.9454;
   DATA[1534,29] := 12.11228;
   DATA[1534,30] := 1.724686;
   DATA[1534,31] := 1.290509;
   DATA[1534,32] := 0.7348846;
   DATA[1534,33] := 0.3082983;
   DATA[1534,34] := 2.0;
   DATA[1534,35] := 250.3365;
   DATA[1534,36] := 1.649953;
   DATA[1534,37] := 189.1022;
   DATA[1534,38] := 0.000128152;
   DATA[1534,39] := 1.0;
   DATA[1535,1] := 814.6125;
   DATA[1535,2] := 1.0;
   DATA[1535,3] := 1.0;
   DATA[1535,4] := 262.6891;
   DATA[1535,5] := 8.46501;
   DATA[1535,6] := 318.8413;
   DATA[1535,8] := 1.0;
   DATA[1535,9] := 1.0;
   DATA[1535,10] := 1.0;
   DATA[1535,11] := 19.81241;
   DATA[1535,12] := 2.213881;
   DATA[1535,13] := 927.8871;
   DATA[1535,14] := 1.0;
   DATA[1535,15] := 2.0;
   DATA[1535,16] := 1.0;
   DATA[1535,17] := 1.0;
   DATA[1535,18] := 1.0;
   DATA[1535,19] := 2.0;
   DATA[1535,20] := 148.808;
   DATA[1535,21] := 153.858;
   DATA[1535,22] := 1.717874;
   DATA[1535,23] := 791.028;
   DATA[1535,24] := 2.0;
   DATA[1535,25] := 2.0;
   DATA[1535,26] := 7.876378;
   DATA[1535,27] := 142.5788;
   DATA[1535,28] := 262.9454;
   DATA[1535,29] := 12.11228;
   DATA[1535,30] := 1.724686;
   DATA[1535,31] := 1.274113;
   DATA[1535,32] := 0.7348846;
   DATA[1535,33] := 0.3082983;
   DATA[1535,34] := 2.0;
   DATA[1535,35] := 250.3365;
   DATA[1535,36] := 1.649953;
   DATA[1535,37] := 189.1983;
   DATA[1535,38] := 0.000128152;
   DATA[1535,39] := 1.0;
   DATA[1536,1] := 814.4162;
   DATA[1536,2] := 1.0;
   DATA[1536,3] := 1.0;
   DATA[1536,4] := 262.6891;
   DATA[1536,5] := 8.46501;
   DATA[1536,6] := 318.8413;
   DATA[1536,8] := 1.0;
   DATA[1536,9] := 1.0;
   DATA[1536,10] := 1.0;
   DATA[1536,11] := 19.83162;
   DATA[1536,12] := 2.213881;
   DATA[1536,13] := 927.5266;
   DATA[1536,14] := 1.0;
   DATA[1536,15] := 2.0;
   DATA[1536,16] := 1.0;
   DATA[1536,17] := 1.0;
   DATA[1536,18] := 1.0;
   DATA[1536,19] := 2.0;
   DATA[1536,20] := 148.808;
   DATA[1536,21] := 153.858;
   DATA[1536,22] := 1.716592;
   DATA[1536,23] := 791.2587;
   DATA[1536,24] := 2.0;
   DATA[1536,25] := 2.0;
   DATA[1536,26] := 7.876378;
   DATA[1536,27] := 142.5788;
   DATA[1536,28] := 262.9454;
   DATA[1536,29] := 12.11228;
   DATA[1536,30] := 1.724814;
   DATA[1536,31] := 1.271935;
   DATA[1536,32] := 0.7348846;
   DATA[1536,33] := 0.3082983;
   DATA[1536,34] := 2.0;
   DATA[1536,35] := 250.3365;
   DATA[1536,36] := 1.649953;
   DATA[1536,37] := 189.1983;
   DATA[1536,38] := 0.000128152;
   DATA[1536,39] := 1.0;
   DATA[1537,1] := 814.377;
   DATA[1537,2] := 1.0;
   DATA[1537,3] := 1.0;
   DATA[1537,4] := 262.6891;
   DATA[1537,5] := 8.46501;
   DATA[1537,6] := 318.8413;
   DATA[1537,8] := 1.0;
   DATA[1537,9] := 1.0;
   DATA[1537,10] := 1.0;
   DATA[1537,11] := 19.83162;
   DATA[1537,12] := 2.213881;
   DATA[1537,13] := 927.086;
   DATA[1537,14] := 1.0;
   DATA[1537,15] := 2.0;
   DATA[1537,16] := 1.0;
   DATA[1537,17] := 1.0;
   DATA[1537,18] := 1.0;
   DATA[1537,19] := 2.0;
   DATA[1537,20] := 148.808;
   DATA[1537,21] := 153.858;
   DATA[1537,22] := 1.715311;
   DATA[1537,23] := 791.1433;
   DATA[1537,24] := 2.0;
   DATA[1537,25] := 2.0;
   DATA[1537,26] := 7.876378;
   DATA[1537,27] := 142.5788;
   DATA[1537,28] := 262.9454;
   DATA[1537,29] := 12.11228;
   DATA[1537,30] := 1.726096;
   DATA[1537,31] := 1.280389;
   DATA[1537,32] := 0.7348846;
   DATA[1537,33] := 0.3082983;
   DATA[1537,34] := 2.0;
   DATA[1537,35] := 250.3365;
   DATA[1537,36] := 1.649953;
   DATA[1537,37] := 189.1983;
   DATA[1537,38] := 0.000128152;
   DATA[1537,39] := 1.0;
   DATA[1538,1] := 814.22;
   DATA[1538,2] := 1.0;
   DATA[1538,3] := 1.0;
   DATA[1538,4] := 262.6891;
   DATA[1538,5] := 8.46501;
   DATA[1538,6] := 318.8413;
   DATA[1538,8] := 1.0;
   DATA[1538,9] := 1.0;
   DATA[1538,10] := 1.0;
   DATA[1538,11] := 19.83162;
   DATA[1538,12] := 2.213881;
   DATA[1538,13] := 926.325;
   DATA[1538,14] := 1.0;
   DATA[1538,15] := 2.0;
   DATA[1538,16] := 1.0;
   DATA[1538,17] := 1.0;
   DATA[1538,18] := 1.0;
   DATA[1538,19] := 2.0;
   DATA[1538,20] := 148.808;
   DATA[1538,21] := 153.858;
   DATA[1538,22] := 1.715311;
   DATA[1538,23] := 791.2971;
   DATA[1538,24] := 2.0;
   DATA[1538,25] := 2.0;
   DATA[1538,26] := 7.876378;
   DATA[1538,27] := 142.5788;
   DATA[1538,28] := 262.9454;
   DATA[1538,29] := 12.11228;
   DATA[1538,30] := 1.726096;
   DATA[1538,31] := 1.284104;
   DATA[1538,32] := 0.736549;
   DATA[1538,33] := 0.3082983;
   DATA[1538,34] := 2.0;
   DATA[1538,35] := 250.3365;
   DATA[1538,36] := 1.649953;
   DATA[1538,37] := 189.1983;
   DATA[1538,38] := 0.000128152;
   DATA[1538,39] := 1.0;
   DATA[1539,1] := 814.2985;
   DATA[1539,2] := 1.0;
   DATA[1539,3] := 1.0;
   DATA[1539,4] := 262.6891;
   DATA[1539,5] := 8.46501;
   DATA[1539,6] := 318.8413;
   DATA[1539,8] := 1.0;
   DATA[1539,9] := 1.0;
   DATA[1539,10] := 1.0;
   DATA[1539,11] := 19.81241;
   DATA[1539,12] := 2.213881;
   DATA[1539,13] := 925.8844;
   DATA[1539,14] := 1.0;
   DATA[1539,15] := 2.0;
   DATA[1539,16] := 1.0;
   DATA[1539,17] := 1.0;
   DATA[1539,18] := 1.0;
   DATA[1539,19] := 2.0;
   DATA[1539,20] := 148.808;
   DATA[1539,21] := 153.858;
   DATA[1539,22] := 1.715311;
   DATA[1539,23] := 791.6047;
   DATA[1539,24] := 2.0;
   DATA[1539,25] := 2.0;
   DATA[1539,26] := 7.876378;
   DATA[1539,27] := 142.5788;
   DATA[1539,28] := 262.9454;
   DATA[1539,29] := 12.11228;
   DATA[1539,30] := 1.726352;
   DATA[1539,31] := 1.291918;
   DATA[1539,32] := 0.7373172;
   DATA[1539,33] := 0.3082983;
   DATA[1539,34] := 2.0;
   DATA[1539,35] := 250.3365;
   DATA[1539,36] := 1.649953;
   DATA[1539,37] := 189.1983;
   DATA[1539,38] := 0.000128152;
   DATA[1539,39] := 1.0;
   DATA[1540,1] := 814.3377;
   DATA[1540,2] := 1.0;
   DATA[1540,3] := 1.0;
   DATA[1540,4] := 262.6891;
   DATA[1540,5] := 8.46501;
   DATA[1540,6] := 318.8413;
   DATA[1540,8] := 1.0;
   DATA[1540,9] := 1.0;
   DATA[1540,10] := 1.0;
   DATA[1540,11] := 19.81241;
   DATA[1540,12] := 2.213881;
   DATA[1540,13] := 925.2435;
   DATA[1540,14] := 1.0;
   DATA[1540,15] := 2.0;
   DATA[1540,16] := 1.0;
   DATA[1540,17] := 1.0;
   DATA[1540,18] := 1.0;
   DATA[1540,19] := 2.0;
   DATA[1540,20] := 148.808;
   DATA[1540,21] := 153.858;
   DATA[1540,22] := 1.715311;
   DATA[1540,23] := 791.2971;
   DATA[1540,24] := 2.0;
   DATA[1540,25] := 2.0;
   DATA[1540,26] := 7.876378;
   DATA[1540,27] := 142.5788;
   DATA[1540,28] := 262.9454;
   DATA[1540,29] := 12.11228;
   DATA[1540,30] := 1.724173;
   DATA[1540,31] := 1.280389;
   DATA[1540,32] := 0.7379573;
   DATA[1540,33] := 0.3082983;
   DATA[1540,34] := 2.0;
   DATA[1540,35] := 250.3365;
   DATA[1540,36] := 1.649953;
   DATA[1540,37] := 189.1983;
   DATA[1540,38] := 0.000128152;
   DATA[1540,39] := 1.0;
   DATA[1541,1] := 814.6125;
   DATA[1541,2] := 1.0;
   DATA[1541,3] := 1.0;
   DATA[1541,4] := 262.6891;
   DATA[1541,5] := 8.46501;
   DATA[1541,6] := 318.8413;
   DATA[1541,8] := 1.0;
   DATA[1541,9] := 1.0;
   DATA[1541,10] := 1.0;
   DATA[1541,11] := 19.81881;
   DATA[1541,12] := 2.213881;
   DATA[1541,13] := 924.4424;
   DATA[1541,14] := 1.0;
   DATA[1541,15] := 2.0;
   DATA[1541,16] := 1.0;
   DATA[1541,17] := 1.0;
   DATA[1541,18] := 1.0;
   DATA[1541,19] := 2.0;
   DATA[1541,20] := 148.808;
   DATA[1541,21] := 153.858;
   DATA[1541,22] := 1.715311;
   DATA[1541,23] := 791.1433;
   DATA[1541,24] := 2.0;
   DATA[1541,25] := 2.0;
   DATA[1541,26] := 7.876378;
   DATA[1541,27] := 142.5788;
   DATA[1541,28] := 262.9454;
   DATA[1541,29] := 12.11228;
   DATA[1541,30] := 1.722123;
   DATA[1541,31] := 1.265787;
   DATA[1541,32] := 0.7379573;
   DATA[1541,33] := 0.3082983;
   DATA[1541,34] := 2.0;
   DATA[1541,35] := 250.3365;
   DATA[1541,36] := 1.649953;
   DATA[1541,37] := 188.9259;
   DATA[1541,38] := 0.000128152;
   DATA[1541,39] := 1.0;
   DATA[1542,1] := 814.6125;
   DATA[1542,2] := 1.0;
   DATA[1542,3] := 1.0;
   DATA[1542,4] := 262.6891;
   DATA[1542,5] := 8.462767;
   DATA[1542,6] := 318.8413;
   DATA[1542,8] := 1.0;
   DATA[1542,9] := 1.0;
   DATA[1542,10] := 1.0;
   DATA[1542,11] := 19.83162;
   DATA[1542,12] := 2.213881;
   DATA[1542,13] := 924.0019;
   DATA[1542,14] := 1.0;
   DATA[1542,15] := 2.0;
   DATA[1542,16] := 1.0;
   DATA[1542,17] := 1.0;
   DATA[1542,18] := 1.0;
   DATA[1542,19] := 2.0;
   DATA[1542,20] := 148.808;
   DATA[1542,21] := 153.858;
   DATA[1542,22] := 1.715311;
   DATA[1542,23] := 791.2971;
   DATA[1542,24] := 2.0;
   DATA[1542,25] := 2.0;
   DATA[1542,26] := 7.876378;
   DATA[1542,27] := 142.5788;
   DATA[1542,28] := 262.9454;
   DATA[1542,29] := 12.11228;
   DATA[1542,30] := 1.722123;
   DATA[1542,31] := 1.261816;
   DATA[1542,32] := 0.7379573;
   DATA[1542,33] := 0.3082983;
   DATA[1542,34] := 2.0;
   DATA[1542,35] := 250.3204;
   DATA[1542,36] := 1.649953;
   DATA[1542,37] := 188.9259;
   DATA[1542,38] := 0.000128152;
   DATA[1542,39] := 1.0;
   DATA[1543,1] := 814.534;
   DATA[1543,2] := 1.0;
   DATA[1543,3] := 1.0;
   DATA[1543,4] := 262.6891;
   DATA[1543,5] := 8.462767;
   DATA[1543,6] := 318.8413;
   DATA[1543,8] := 1.0;
   DATA[1543,9] := 1.0;
   DATA[1543,10] := 1.0;
   DATA[1543,11] := 19.85402;
   DATA[1543,12] := 2.213881;
   DATA[1543,13] := 923.6815;
   DATA[1543,14] := 1.0;
   DATA[1543,15] := 2.0;
   DATA[1543,16] := 1.0;
   DATA[1543,17] := 1.0;
   DATA[1543,18] := 1.0;
   DATA[1543,19] := 2.0;
   DATA[1543,20] := 148.808;
   DATA[1543,21] := 153.858;
   DATA[1543,22] := 1.711723;
   DATA[1543,23] := 791.6047;
   DATA[1543,24] := 2.0;
   DATA[1543,25] := 2.0;
   DATA[1543,26] := 7.876378;
   DATA[1543,27] := 142.5788;
   DATA[1543,28] := 262.9454;
   DATA[1543,29] := 12.11228;
   DATA[1543,30] := 1.722123;
   DATA[1543,31] := 1.261176;
   DATA[1543,32] := 0.7379573;
   DATA[1543,33] := 0.3082983;
   DATA[1543,34] := 2.0;
   DATA[1543,35] := 250.1122;
   DATA[1543,36] := 1.649953;
   DATA[1543,37] := 188.9259;
   DATA[1543,38] := 0.000128152;
   DATA[1543,39] := 1.0;
   DATA[1544,1] := 814.5732;
   DATA[1544,2] := 1.0;
   DATA[1544,3] := 1.0;
   DATA[1544,4] := 262.6891;
   DATA[1544,5] := 8.462767;
   DATA[1544,6] := 318.8413;
   DATA[1544,8] := 1.0;
   DATA[1544,9] := 1.0;
   DATA[1544,10] := 1.0;
   DATA[1544,11] := 19.76759;
   DATA[1544,12] := 2.216058;
   DATA[1544,13] := 923.1207;
   DATA[1544,14] := 1.0;
   DATA[1544,15] := 2.0;
   DATA[1544,16] := 1.0;
   DATA[1544,17] := 1.0;
   DATA[1544,18] := 1.0;
   DATA[1544,19] := 2.0;
   DATA[1544,20] := 148.808;
   DATA[1544,21] := 153.858;
   DATA[1544,22] := 1.711723;
   DATA[1544,23] := 791.2971;
   DATA[1544,24] := 2.0;
   DATA[1544,25] := 2.0;
   DATA[1544,26] := 7.876378;
   DATA[1544,27] := 142.6557;
   DATA[1544,28] := 262.9454;
   DATA[1544,29] := 12.11228;
   DATA[1544,30] := 1.723661;
   DATA[1544,31] := 1.261176;
   DATA[1544,32] := 0.7352687;
   DATA[1544,33] := 0.3082983;
   DATA[1544,34] := 2.0;
   DATA[1544,35] := 250.1122;
   DATA[1544,36] := 1.649953;
   DATA[1544,37] := 188.9259;
   DATA[1544,38] := 0.000128152;
   DATA[1544,39] := 1.0;
   DATA[1545,1] := 814.534;
   DATA[1545,2] := 1.0;
   DATA[1545,3] := 1.0;
   DATA[1545,4] := 262.6891;
   DATA[1545,5] := 8.462767;
   DATA[1545,6] := 318.8413;
   DATA[1545,8] := 1.0;
   DATA[1545,9] := 1.0;
   DATA[1545,10] := 1.0;
   DATA[1545,11] := 19.74838;
   DATA[1545,12] := 2.216058;
   DATA[1545,13] := 922.8403;
   DATA[1545,14] := 1.0;
   DATA[1545,15] := 2.0;
   DATA[1545,16] := 1.0;
   DATA[1545,17] := 1.0;
   DATA[1545,18] := 1.0;
   DATA[1545,19] := 2.0;
   DATA[1545,20] := 148.808;
   DATA[1545,21] := 153.858;
   DATA[1545,22] := 1.713517;
   DATA[1545,23] := 791.6816;
   DATA[1545,24] := 2.0;
   DATA[1545,25] := 2.0;
   DATA[1545,26] := 7.876378;
   DATA[1545,27] := 142.6814;
   DATA[1545,28] := 262.9454;
   DATA[1545,29] := 12.11228;
   DATA[1545,30] := 1.724814;
   DATA[1545,31] := 1.276547;
   DATA[1545,32] := 0.7352687;
   DATA[1545,33] := 0.3082983;
   DATA[1545,34] := 2.0;
   DATA[1545,35] := 250.1122;
   DATA[1545,36] := 1.649953;
   DATA[1545,37] := 188.9259;
   DATA[1545,38] := 0.000128152;
   DATA[1545,39] := 1.0;
   DATA[1546,1] := 814.534;
   DATA[1546,2] := 1.0;
   DATA[1546,3] := 1.0;
   DATA[1546,4] := 262.6891;
   DATA[1546,5] := 8.462767;
   DATA[1546,6] := 318.8413;
   DATA[1546,8] := 1.0;
   DATA[1546,9] := 1.0;
   DATA[1546,10] := 1.0;
   DATA[1546,11] := 19.74838;
   DATA[1546,12] := 2.214137;
   DATA[1546,13] := 922.1193;
   DATA[1546,14] := 1.0;
   DATA[1546,15] := 2.0;
   DATA[1546,16] := 1.0;
   DATA[1546,17] := 1.0;
   DATA[1546,18] := 1.0;
   DATA[1546,19] := 2.0;
   DATA[1546,20] := 148.808;
   DATA[1546,21] := 153.858;
   DATA[1546,22] := 1.714542;
   DATA[1546,23] := 791.8354;
   DATA[1546,24] := 2.0;
   DATA[1546,25] := 2.0;
   DATA[1546,26] := 7.876378;
   DATA[1546,27] := 142.6814;
   DATA[1546,28] := 262.9454;
   DATA[1546,29] := 12.11228;
   DATA[1546,30] := 1.724814;
   DATA[1546,31] := 1.28103;
   DATA[1546,32] := 0.7352687;
   DATA[1546,33] := 0.3082983;
   DATA[1546,34] := 2.0;
   DATA[1546,35] := 250.1122;
   DATA[1546,36] := 1.649953;
   DATA[1546,37] := 189.0541;
   DATA[1546,38] := 0.000128152;
   DATA[1546,39] := 1.0;
   DATA[1547,1] := 814.8873;
   DATA[1547,2] := 1.0;
   DATA[1547,3] := 1.0;
   DATA[1547,4] := 262.6891;
   DATA[1547,5] := 8.463408;
   DATA[1547,6] := 318.8413;
   DATA[1547,8] := 1.0;
   DATA[1547,9] := 1.0;
   DATA[1547,10] := 1.0;
   DATA[1547,11] := 19.70037;
   DATA[1547,12] := 2.213881;
   DATA[1547,13] := 921.9191;
   DATA[1547,14] := 1.0;
   DATA[1547,15] := 2.0;
   DATA[1547,16] := 1.0;
   DATA[1547,17] := 1.0;
   DATA[1547,18] := 1.0;
   DATA[1547,19] := 2.0;
   DATA[1547,20] := 148.808;
   DATA[1547,21] := 153.6529;
   DATA[1547,22] := 1.714542;
   DATA[1547,23] := 792.1046;
   DATA[1547,24] := 2.0;
   DATA[1547,25] := 2.0;
   DATA[1547,26] := 7.876378;
   DATA[1547,27] := 142.6814;
   DATA[1547,28] := 262.9454;
   DATA[1547,29] := 12.11228;
   DATA[1547,30] := 1.724814;
   DATA[1547,31] := 1.275394;
   DATA[1547,32] := 0.7352687;
   DATA[1547,33] := 0.3082983;
   DATA[1547,34] := 2.0;
   DATA[1547,35] := 250.1122;
   DATA[1547,36] := 1.649953;
   DATA[1547,37] := 189.0541;
   DATA[1547,38] := 0.000128152;
   DATA[1547,39] := 1.0;
   DATA[1548,1] := 814.7695;
   DATA[1548,2] := 1.0;
   DATA[1548,3] := 1.0;
   DATA[1548,4] := 262.6891;
   DATA[1548,5] := 8.463728;
   DATA[1548,6] := 318.8413;
   DATA[1548,8] := 1.0;
   DATA[1548,9] := 1.0;
   DATA[1548,10] := 1.0;
   DATA[1548,11] := 19.70037;
   DATA[1548,12] := 2.213881;
   DATA[1548,13] := 921.2782;
   DATA[1548,14] := 1.0;
   DATA[1548,15] := 2.0;
   DATA[1548,16] := 1.0;
   DATA[1548,17] := 1.0;
   DATA[1548,18] := 1.0;
   DATA[1548,19] := 2.0;
   DATA[1548,20] := 148.808;
   DATA[1548,21] := 153.6529;
   DATA[1548,22] := 1.71467;
   DATA[1548,23] := 792.1815;
   DATA[1548,24] := 2.0;
   DATA[1548,25] := 2.0;
   DATA[1548,26] := 7.876378;
   DATA[1548,27] := 142.6814;
   DATA[1548,28] := 262.9454;
   DATA[1548,29] := 12.11228;
   DATA[1548,30] := 1.724814;
   DATA[1548,31] := 1.28103;
   DATA[1548,32] := 0.7352687;
   DATA[1548,33] := 0.3082983;
   DATA[1548,34] := 2.0;
   DATA[1548,35] := 250.3365;
   DATA[1548,36] := 1.649953;
   DATA[1548,37] := 189.0541;
   DATA[1548,38] := 0.000128152;
   DATA[1548,39] := 1.0;
   DATA[1549,1] := 814.7695;
   DATA[1549,2] := 1.0;
   DATA[1549,3] := 1.0;
   DATA[1549,4] := 262.6891;
   DATA[1549,5] := 8.463728;
   DATA[1549,6] := 318.8413;
   DATA[1549,8] := 1.0;
   DATA[1549,9] := 1.0;
   DATA[1549,10] := 1.0;
   DATA[1549,11] := 19.70037;
   DATA[1549,12] := 2.213881;
   DATA[1549,13] := 920.8376;
   DATA[1549,14] := 1.0;
   DATA[1549,15] := 2.0;
   DATA[1549,16] := 1.0;
   DATA[1549,17] := 1.0;
   DATA[1549,18] := 1.0;
   DATA[1549,19] := 2.0;
   DATA[1549,20] := 148.808;
   DATA[1549,21] := 153.6529;
   DATA[1549,22] := 1.715567;
   DATA[1549,23] := 792.1815;
   DATA[1549,24] := 2.0;
   DATA[1549,25] := 2.0;
   DATA[1549,26] := 7.876378;
   DATA[1549,27] := 142.6814;
   DATA[1549,28] := 262.9454;
   DATA[1549,29] := 12.11228;
   DATA[1549,30] := 1.724814;
   DATA[1549,31] := 1.286922;
   DATA[1549,32] := 0.7352687;
   DATA[1549,33] := 0.3082983;
   DATA[1549,34] := 2.0;
   DATA[1549,35] := 250.3365;
   DATA[1549,36] := 1.649953;
   DATA[1549,37] := 189.1342;
   DATA[1549,38] := 0.000128152;
   DATA[1549,39] := 1.0;
   DATA[1550,1] := 814.9658;
   DATA[1550,2] := 1.0;
   DATA[1550,3] := 1.0;
   DATA[1550,4] := 262.5288;
   DATA[1550,5] := 8.464369;
   DATA[1550,6] := 318.8413;
   DATA[1550,8] := 1.0;
   DATA[1550,9] := 1.0;
   DATA[1550,10] := 1.0;
   DATA[1550,11] := 19.7836;
   DATA[1550,12] := 2.213881;
   DATA[1550,13] := 920.2368;
   DATA[1550,14] := 1.0;
   DATA[1550,15] := 2.0;
   DATA[1550,16] := 1.0;
   DATA[1550,17] := 1.0;
   DATA[1550,18] := 1.0;
   DATA[1550,19] := 2.0;
   DATA[1550,20] := 148.808;
   DATA[1550,21] := 153.8067;
   DATA[1550,22] := 1.715567;
   DATA[1550,23] := 792.1815;
   DATA[1550,24] := 2.0;
   DATA[1550,25] := 2.0;
   DATA[1550,26] := 7.876378;
   DATA[1550,27] := 142.6814;
   DATA[1550,28] := 262.9454;
   DATA[1550,29] := 12.11228;
   DATA[1550,30] := 1.725711;
   DATA[1550,31] := 1.298322;
   DATA[1550,32] := 0.7352687;
   DATA[1550,33] := 0.3082983;
   DATA[1550,34] := 2.0;
   DATA[1550,35] := 250.3365;
   DATA[1550,36] := 1.649953;
   DATA[1550,37] := 189.1342;
   DATA[1550,38] := 0.000128152;
   DATA[1550,39] := 1.0;
   DATA[1551,1] := 815.319;
   DATA[1551,2] := 1.0;
   DATA[1551,3] := 1.0;
   DATA[1551,4] := 262.5288;
   DATA[1551,5] := 8.464369;
   DATA[1551,6] := 318.9695;
   DATA[1551,8] := 1.0;
   DATA[1551,9] := 1.0;
   DATA[1551,10] := 1.0;
   DATA[1551,11] := 19.7836;
   DATA[1551,12] := 2.213881;
   DATA[1551,13] := 920.0766;
   DATA[1551,14] := 1.0;
   DATA[1551,15] := 2.0;
   DATA[1551,16] := 1.0;
   DATA[1551,17] := 1.0;
   DATA[1551,18] := 1.0;
   DATA[1551,19] := 2.0;
   DATA[1551,20] := 148.808;
   DATA[1551,21] := 153.8067;
   DATA[1551,22] := 1.715567;
   DATA[1551,23] := 791.9124;
   DATA[1551,24] := 2.0;
   DATA[1551,25] := 2.0;
   DATA[1551,26] := 7.876378;
   DATA[1551,27] := 142.6814;
   DATA[1551,28] := 262.9454;
   DATA[1551,29] := 12.11228;
   DATA[1551,30] := 1.726993;
   DATA[1551,31] := 1.301524;
   DATA[1551,32] := 0.7352687;
   DATA[1551,33] := 0.3082983;
   DATA[1551,34] := 2.0;
   DATA[1551,35] := 250.3365;
   DATA[1551,36] := 1.649953;
   DATA[1551,37] := 189.1342;
   DATA[1551,38] := 0.000128152;
   DATA[1551,39] := 1.0;
   DATA[1552,1] := 815.1228;
   DATA[1552,2] := 1.0;
   DATA[1552,3] := 1.0;
   DATA[1552,4] := 262.5288;
   DATA[1552,5] := 8.464369;
   DATA[1552,6] := 318.9695;
   DATA[1552,8] := 1.0;
   DATA[1552,9] := 1.0;
   DATA[1552,10] := 1.0;
   DATA[1552,11] := 19.74198;
   DATA[1552,12] := 2.215418;
   DATA[1552,13] := 919.5159;
   DATA[1552,14] := 1.0;
   DATA[1552,15] := 2.0;
   DATA[1552,16] := 1.0;
   DATA[1552,17] := 1.0;
   DATA[1552,18] := 1.0;
   DATA[1552,19] := 2.0;
   DATA[1552,20] := 148.808;
   DATA[1552,21] := 153.8067;
   DATA[1552,22] := 1.715567;
   DATA[1552,23] := 791.797;
   DATA[1552,24] := 2.0;
   DATA[1552,25] := 2.0;
   DATA[1552,26] := 7.876378;
   DATA[1552,27] := 142.6814;
   DATA[1552,28] := 262.9454;
   DATA[1552,29] := 12.11228;
   DATA[1552,30] := 1.726993;
   DATA[1552,31] := 1.301524;
   DATA[1552,32] := 0.7352687;
   DATA[1552,33] := 0.3082983;
   DATA[1552,34] := 2.0;
   DATA[1552,35] := 250.3365;
   DATA[1552,36] := 1.649953;
   DATA[1552,37] := 189.1342;
   DATA[1552,38] := 0.000128152;
   DATA[1552,39] := 1.0;
   DATA[1553,1] := 815.5153;
   DATA[1553,2] := 1.0;
   DATA[1553,3] := 1.0;
   DATA[1553,4] := 262.5288;
   DATA[1553,5] := 8.464369;
   DATA[1553,6] := 318.9695;
   DATA[1553,8] := 1.0;
   DATA[1553,9] := 1.0;
   DATA[1553,10] := 1.0;
   DATA[1553,11] := 19.70357;
   DATA[1553,12] := 2.216187;
   DATA[1553,13] := 918.835;
   DATA[1553,14] := 1.0;
   DATA[1553,15] := 2.0;
   DATA[1553,16] := 1.0;
   DATA[1553,17] := 1.0;
   DATA[1553,18] := 1.0;
   DATA[1553,19] := 2.0;
   DATA[1553,20] := 148.808;
   DATA[1553,21] := 153.8067;
   DATA[1553,22] := 1.715567;
   DATA[1553,23] := 792.4891;
   DATA[1553,24] := 2.0;
   DATA[1553,25] := 2.0;
   DATA[1553,26] := 7.876378;
   DATA[1553,27] := 142.6814;
   DATA[1553,28] := 262.9454;
   DATA[1553,29] := 12.11228;
   DATA[1553,30] := 1.726993;
   DATA[1553,31] := 1.291277;
   DATA[1553,32] := 0.7352687;
   DATA[1553,33] := 0.3082983;
   DATA[1553,34] := 2.0;
   DATA[1553,35] := 250.3365;
   DATA[1553,36] := 1.649953;
   DATA[1553,37] := 189.1342;
   DATA[1553,38] := 0.000128152;
   DATA[1553,39] := 1.0;
   DATA[1554,1] := 815.5546;
   DATA[1554,2] := 1.0;
   DATA[1554,3] := 1.0;
   DATA[1554,4] := 262.5288;
   DATA[1554,5] := 8.464369;
   DATA[1554,6] := 318.9695;
   DATA[1554,8] := 1.0;
   DATA[1554,9] := 1.0;
   DATA[1554,10] := 1.0;
   DATA[1554,11] := 19.63634;
   DATA[1554,12] := 2.216187;
   DATA[1554,13] := 918.7148;
   DATA[1554,14] := 1.0;
   DATA[1554,15] := 2.0;
   DATA[1554,16] := 1.0;
   DATA[1554,17] := 1.0;
   DATA[1554,18] := 1.0;
   DATA[1554,19] := 2.0;
   DATA[1554,20] := 148.808;
   DATA[1554,21] := 153.8067;
   DATA[1554,22] := 1.714926;
   DATA[1554,23] := 792.6044;
   DATA[1554,24] := 2.0;
   DATA[1554,25] := 2.0;
   DATA[1554,26] := 7.876378;
   DATA[1554,27] := 142.6814;
   DATA[1554,28] := 262.9454;
   DATA[1554,29] := 12.11228;
   DATA[1554,30] := 1.725583;
   DATA[1554,31] := 1.291277;
   DATA[1554,32] := 0.7352687;
   DATA[1554,33] := 0.3082983;
   DATA[1554,34] := 2.0;
   DATA[1554,35] := 250.3365;
   DATA[1554,36] := 1.762086;
   DATA[1554,37] := 189.1342;
   DATA[1554,38] := 0.000128152;
   DATA[1554,39] := 1.0;
   DATA[1555,1] := 815.5546;
   DATA[1555,2] := 1.0;
   DATA[1555,3] := 1.0;
   DATA[1555,4] := 262.5288;
   DATA[1555,5] := 8.464369;
   DATA[1555,6] := 318.9695;
   DATA[1555,8] := 1.0;
   DATA[1555,9] := 1.0;
   DATA[1555,10] := 1.0;
   DATA[1555,11] := 19.63634;
   DATA[1555,12] := 2.216187;
   DATA[1555,13] := 918.7148;
   DATA[1555,14] := 1.0;
   DATA[1555,15] := 2.0;
   DATA[1555,16] := 1.0;
   DATA[1555,17] := 1.0;
   DATA[1555,18] := 1.0;
   DATA[1555,19] := 2.0;
   DATA[1555,20] := 148.808;
   DATA[1555,21] := 153.8067;
   DATA[1555,22] := 1.714926;
   DATA[1555,23] := 792.6044;
   DATA[1555,24] := 2.0;
   DATA[1555,25] := 2.0;
   DATA[1555,26] := 7.876378;
   DATA[1555,27] := 142.6814;
   DATA[1555,28] := 262.9454;
   DATA[1555,29] := 12.11228;
   DATA[1555,30] := 1.725583;
   DATA[1555,31] := 1.291277;
   DATA[1555,32] := 0.7352687;
   DATA[1555,33] := 0.3082983;
   DATA[1555,34] := 2.0;
   DATA[1555,35] := 250.3365;
   DATA[1555,36] := 1.762086;
   DATA[1555,37] := 189.1342;
   DATA[1555,38] := 0.000128152;
   DATA[1555,39] := 1.0;
   DATA[1556,1] := 815.5153;
   DATA[1556,2] := 1.0;
   DATA[1556,3] := 1.0;
   DATA[1556,4] := 262.5288;
   DATA[1556,5] := 8.464369;
   DATA[1556,6] := 318.9695;
   DATA[1556,8] := 1.0;
   DATA[1556,9] := 1.0;
   DATA[1556,10] := 1.0;
   DATA[1556,11] := 19.63634;
   DATA[1556,12] := 2.216187;
   DATA[1556,13] := 918.2341;
   DATA[1556,14] := 1.0;
   DATA[1556,15] := 2.0;
   DATA[1556,16] := 1.0;
   DATA[1556,17] := 1.0;
   DATA[1556,18] := 1.0;
   DATA[1556,19] := 2.0;
   DATA[1556,20] := 148.808;
   DATA[1556,21] := 153.8067;
   DATA[1556,22] := 1.714926;
   DATA[1556,23] := 792.4122;
   DATA[1556,24] := 2.0;
   DATA[1556,25] := 2.0;
   DATA[1556,26] := 7.876378;
   DATA[1556,27] := 142.6814;
   DATA[1556,28] := 262.9454;
   DATA[1556,29] := 12.11228;
   DATA[1556,30] := 1.725455;
   DATA[1556,31] := 1.288203;
   DATA[1556,32] := 0.7352687;
   DATA[1556,33] := 0.3082983;
   DATA[1556,34] := 2.0;
   DATA[1556,35] := 250.1923;
   DATA[1556,36] := 1.762086;
   DATA[1556,37] := 189.0541;
   DATA[1556,38] := 0.000128152;
   DATA[1556,39] := 1.0;
   DATA[1557,1] := 815.319;
   DATA[1557,2] := 1.0;
   DATA[1557,3] := 1.0;
   DATA[1557,4] := 262.5288;
   DATA[1557,5] := 8.464369;
   DATA[1557,6] := 318.9695;
   DATA[1557,8] := 1.0;
   DATA[1557,9] := 1.0;
   DATA[1557,10] := 1.0;
   DATA[1557,11] := 19.63634;
   DATA[1557,12] := 2.216187;
   DATA[1557,13] := 917.6333;
   DATA[1557,14] := 1.0;
   DATA[1557,15] := 2.0;
   DATA[1557,16] := 1.0;
   DATA[1557,17] := 1.0;
   DATA[1557,18] := 1.0;
   DATA[1557,19] := 2.0;
   DATA[1557,20] := 148.808;
   DATA[1557,21] := 153.8067;
   DATA[1557,22] := 1.714926;
   DATA[1557,23] := 792.7967;
   DATA[1557,24] := 2.0;
   DATA[1557,25] := 2.0;
   DATA[1557,26] := 7.876378;
   DATA[1557,27] := 142.6814;
   DATA[1557,28] := 262.9454;
   DATA[1557,29] := 12.11228;
   DATA[1557,30] := 1.725455;
   DATA[1557,31] := 1.273985;
   DATA[1557,32] := 0.7352687;
   DATA[1557,33] := 0.3082983;
   DATA[1557,34] := 2.0;
   DATA[1557,35] := 250.1602;
   DATA[1557,36] := 1.762086;
   DATA[1557,37] := 189.006;
   DATA[1557,38] := 0.000128152;
   DATA[1557,39] := 1.0;
   DATA[1558,1] := 815.7508;
   DATA[1558,2] := 1.0;
   DATA[1558,3] := 1.0;
   DATA[1558,4] := 262.5288;
   DATA[1558,5] := 8.464369;
   DATA[1558,6] := 318.9695;
   DATA[1558,8] := 1.0;
   DATA[1558,9] := 1.0;
   DATA[1558,10] := 1.0;
   DATA[1558,11] := 19.66835;
   DATA[1558,12] := 2.216187;
   DATA[1558,13] := 917.5132;
   DATA[1558,14] := 1.0;
   DATA[1558,15] := 2.0;
   DATA[1558,16] := 1.0;
   DATA[1558,17] := 1.0;
   DATA[1558,18] := 1.0;
   DATA[1558,19] := 2.0;
   DATA[1558,20] := 148.808;
   DATA[1558,21] := 153.8067;
   DATA[1558,22] := 1.713517;
   DATA[1558,23] := 792.6429;
   DATA[1558,24] := 2.0;
   DATA[1558,25] := 2.0;
   DATA[1558,26] := 7.876378;
   DATA[1558,27] := 142.6814;
   DATA[1558,28] := 262.9454;
   DATA[1558,29] := 12.11228;
   DATA[1558,30] := 1.72443;
   DATA[1558,31] := 1.271295;
   DATA[1558,32] := 0.7352687;
   DATA[1558,33] := 0.3082983;
   DATA[1558,34] := 2.0;
   DATA[1558,35] := 250.1602;
   DATA[1558,36] := 1.649953;
   DATA[1558,37] := 189.006;
   DATA[1558,38] := 0.000128152;
   DATA[1558,39] := 1.0;
   DATA[1559,1] := 815.7115;
   DATA[1559,2] := 1.0;
   DATA[1559,3] := 1.0;
   DATA[1559,4] := 262.5288;
   DATA[1559,5] := 8.464369;
   DATA[1559,6] := 318.9695;
   DATA[1559,8] := 1.0;
   DATA[1559,9] := 1.0;
   DATA[1559,10] := 1.0;
   DATA[1559,11] := 19.71957;
   DATA[1559,12] := 2.214009;
   DATA[1559,13] := 917.0325;
   DATA[1559,14] := 1.0;
   DATA[1559,15] := 2.0;
   DATA[1559,16] := 1.0;
   DATA[1559,17] := 1.0;
   DATA[1559,18] := 1.0;
   DATA[1559,19] := 2.0;
   DATA[1559,20] := 148.808;
   DATA[1559,21] := 153.8067;
   DATA[1559,22] := 1.712748;
   DATA[1559,23] := 792.6813;
   DATA[1559,24] := 2.0;
   DATA[1559,25] := 2.0;
   DATA[1559,26] := 7.876378;
   DATA[1559,27] := 142.6814;
   DATA[1559,28] := 262.9454;
   DATA[1559,29] := 12.11228;
   DATA[1559,30] := 1.72302;
   DATA[1559,31] := 1.271295;
   DATA[1559,32] := 0.7352687;
   DATA[1559,33] := 0.3082983;
   DATA[1559,34] := 2.0;
   DATA[1559,35] := 250.1602;
   DATA[1559,36] := 1.649953;
   DATA[1559,37] := 189.006;
   DATA[1559,38] := 0.000128152;
   DATA[1559,39] := 1.0;
   DATA[1560,1] := 815.7508;
   DATA[1560,2] := 1.0;
   DATA[1560,3] := 1.0;
   DATA[1560,4] := 262.5288;
   DATA[1560,5] := 8.464369;
   DATA[1560,6] := 318.9695;
   DATA[1560,8] := 1.0;
   DATA[1560,9] := 1.0;
   DATA[1560,10] := 1.0;
   DATA[1560,11] := 19.74838;
   DATA[1560,12] := 2.214009;
   DATA[1560,13] := 916.3917;
   DATA[1560,14] := 1.0;
   DATA[1560,15] := 2.0;
   DATA[1560,16] := 1.0;
   DATA[1560,17] := 1.0;
   DATA[1560,18] := 1.0;
   DATA[1560,19] := 2.0;
   DATA[1560,20] := 148.808;
   DATA[1560,21] := 153.8067;
   DATA[1560,22] := 1.712748;
   DATA[1560,23] := 792.7967;
   DATA[1560,24] := 2.0;
   DATA[1560,25] := 2.0;
   DATA[1560,26] := 7.876378;
   DATA[1560,27] := 142.6814;
   DATA[1560,28] := 262.9454;
   DATA[1560,29] := 12.11228;
   DATA[1560,30] := 1.72302;
   DATA[1560,31] := 1.273216;
   DATA[1560,32] := 0.7352687;
   DATA[1560,33] := 0.3082983;
   DATA[1560,34] := 2.0;
   DATA[1560,35] := 250.1602;
   DATA[1560,36] := 1.649953;
   DATA[1560,37] := 189.006;
   DATA[1560,38] := 0.000128152;
   DATA[1560,39] := 1.0;
   DATA[1561,1] := 815.3975;
   DATA[1561,2] := 1.0;
   DATA[1561,3] := 1.0;
   DATA[1561,4] := 262.5288;
   DATA[1561,5] := 8.464369;
   DATA[1561,6] := 318.9695;
   DATA[1561,8] := 1.0;
   DATA[1561,9] := 1.0;
   DATA[1561,10] := 1.0;
   DATA[1561,11] := 19.74838;
   DATA[1561,12] := 2.212343;
   DATA[1561,13] := 916.3917;
   DATA[1561,14] := 1.0;
   DATA[1561,15] := 2.0;
   DATA[1561,16] := 1.0;
   DATA[1561,17] := 1.0;
   DATA[1561,18] := 1.0;
   DATA[1561,19] := 2.0;
   DATA[1561,20] := 148.808;
   DATA[1561,21] := 153.8067;
   DATA[1561,22] := 1.714286;
   DATA[1561,23] := 793.2197;
   DATA[1561,24] := 2.0;
   DATA[1561,25] := 2.0;
   DATA[1561,26] := 7.876378;
   DATA[1561,27] := 142.6814;
   DATA[1561,28] := 262.9454;
   DATA[1561,29] := 12.11228;
   DATA[1561,30] := 1.72302;
   DATA[1561,31] := 1.281286;
   DATA[1561,32] := 0.7352687;
   DATA[1561,33] := 0.3082983;
   DATA[1561,34] := 2.0;
   DATA[1561,35] := 250.0;
   DATA[1561,36] := 1.649953;
   DATA[1561,37] := 188.8138;
   DATA[1561,38] := 0.000128152;
   DATA[1561,39] := 1.0;
   DATA[1562,1] := 815.0835;
   DATA[1562,2] := 1.0;
   DATA[1562,3] := 1.0;
   DATA[1562,4] := 262.5288;
   DATA[1562,5] := 8.464369;
   DATA[1562,6] := 318.9695;
   DATA[1562,8] := 1.0;
   DATA[1562,9] := 1.0;
   DATA[1562,10] := 1.0;
   DATA[1562,11] := 19.74838;
   DATA[1562,12] := 2.212343;
   DATA[1562,13] := 915.8309;
   DATA[1562,14] := 1.0;
   DATA[1562,15] := 2.0;
   DATA[1562,16] := 1.0;
   DATA[1562,17] := 1.0;
   DATA[1562,18] := 1.0;
   DATA[1562,19] := 2.0;
   DATA[1562,20] := 148.808;
   DATA[1562,21] := 153.6785;
   DATA[1562,22] := 1.714542;
   DATA[1562,23] := 793.4119;
   DATA[1562,24] := 2.0;
   DATA[1562,25] := 2.0;
   DATA[1562,26] := 7.876378;
   DATA[1562,27] := 142.6814;
   DATA[1562,28] := 262.9454;
   DATA[1562,29] := 12.11228;
   DATA[1562,30] := 1.72302;
   DATA[1562,31] := 1.291149;
   DATA[1562,32] := 0.7352687;
   DATA[1562,33] := 0.3082983;
   DATA[1562,34] := 2.0;
   DATA[1562,35] := 249.984;
   DATA[1562,36] := 1.649953;
   DATA[1562,37] := 188.8138;
   DATA[1562,38] := 0.000128152;
   DATA[1562,39] := 1.0;
   DATA[1563,1] := 815.319;
   DATA[1563,2] := 1.0;
   DATA[1563,3] := 1.0;
   DATA[1563,4] := 262.5288;
   DATA[1563,5] := 8.464369;
   DATA[1563,6] := 318.9695;
   DATA[1563,8] := 1.0;
   DATA[1563,9] := 1.0;
   DATA[1563,10] := 1.0;
   DATA[1563,11] := 19.74838;
   DATA[1563,12] := 2.210806;
   DATA[1563,13] := 915.1901;
   DATA[1563,14] := 1.0;
   DATA[1563,15] := 2.0;
   DATA[1563,16] := 1.0;
   DATA[1563,17] := 1.0;
   DATA[1563,18] := 1.0;
   DATA[1563,19] := 2.0;
   DATA[1563,20] := 148.808;
   DATA[1563,21] := 153.6785;
   DATA[1563,22] := 1.714542;
   DATA[1563,23] := 793.5657;
   DATA[1563,24] := 2.0;
   DATA[1563,25] := 2.0;
   DATA[1563,26] := 7.876378;
   DATA[1563,27] := 142.8608;
   DATA[1563,28] := 262.8493;
   DATA[1563,29] := 12.11228;
   DATA[1563,30] := 1.72302;
   DATA[1563,31] := 1.292046;
   DATA[1563,32] := 0.7352687;
   DATA[1563,33] := 0.3086827;
   DATA[1563,34] := 2.0;
   DATA[1563,35] := 249.984;
   DATA[1563,36] := 1.649953;
   DATA[1563,37] := 188.8138;
   DATA[1563,38] := 0.000128152;
   DATA[1563,39] := 1.0;
   DATA[1564,1] := 815.5153;
   DATA[1564,2] := 1.0;
   DATA[1564,3] := 1.0;
   DATA[1564,4] := 262.5288;
   DATA[1564,5] := 8.464369;
   DATA[1564,6] := 318.9695;
   DATA[1564,8] := 1.0;
   DATA[1564,9] := 1.0;
   DATA[1564,10] := 1.0;
   DATA[1564,11] := 19.74838;
   DATA[1564,12] := 2.21055;
   DATA[1564,13] := 915.1901;
   DATA[1564,14] := 1.0;
   DATA[1564,15] := 2.0;
   DATA[1564,16] := 1.0;
   DATA[1564,17] := 1.0;
   DATA[1564,18] := 1.0;
   DATA[1564,19] := 2.0;
   DATA[1564,20] := 148.808;
   DATA[1564,21] := 153.6785;
   DATA[1564,22] := 1.714542;
   DATA[1564,23] := 793.6042;
   DATA[1564,24] := 2.0;
   DATA[1564,25] := 2.0;
   DATA[1564,26] := 7.876378;
   DATA[1564,27] := 142.8608;
   DATA[1564,28] := 262.8172;
   DATA[1564,29] := 12.11228;
   DATA[1564,30] := 1.722763;
   DATA[1564,31] := 1.292046;
   DATA[1564,32] := 0.7352687;
   DATA[1564,33] := 0.3086827;
   DATA[1564,34] := 2.0;
   DATA[1564,35] := 249.984;
   DATA[1564,36] := 1.649953;
   DATA[1564,37] := 188.8138;
   DATA[1564,38] := 0.000128152;
   DATA[1564,39] := 1.0;
   DATA[1565,1] := 815.0835;
   DATA[1565,2] := 1.0;
   DATA[1565,3] := 1.0;
   DATA[1565,4] := 262.5288;
   DATA[1565,5] := 8.464369;
   DATA[1565,6] := 318.9695;
   DATA[1565,8] := 1.0;
   DATA[1565,9] := 1.0;
   DATA[1565,10] := 1.0;
   DATA[1565,11] := 19.74838;
   DATA[1565,12] := 2.21055;
   DATA[1565,13] := 914.6693;
   DATA[1565,14] := 1.0;
   DATA[1565,15] := 2.0;
   DATA[1565,16] := 1.0;
   DATA[1565,17] := 1.0;
   DATA[1565,18] := 1.0;
   DATA[1565,19] := 2.0;
   DATA[1565,20] := 148.808;
   DATA[1565,21] := 153.6785;
   DATA[1565,22] := 1.71262;
   DATA[1565,23] := 793.8349;
   DATA[1565,24] := 2.0;
   DATA[1565,25] := 2.0;
   DATA[1565,26] := 7.876378;
   DATA[1565,27] := 142.8608;
   DATA[1565,28] := 262.8172;
   DATA[1565,29] := 12.11228;
   DATA[1565,30] := 1.722251;
   DATA[1565,31] := 1.298834;
   DATA[1565,32] := 0.7352687;
   DATA[1565,33] := 0.3086827;
   DATA[1565,34] := 2.0;
   DATA[1565,35] := 249.984;
   DATA[1565,36] := 1.649953;
   DATA[1565,37] := 188.8138;
   DATA[1565,38] := 0.000128152;
   DATA[1565,39] := 1.0;
   DATA[1566,1] := 815.0835;
   DATA[1566,2] := 1.0;
   DATA[1566,3] := 1.0;
   DATA[1566,4] := 262.5288;
   DATA[1566,5] := 8.464369;
   DATA[1566,6] := 318.9695;
   DATA[1566,8] := 1.0;
   DATA[1566,9] := 1.0;
   DATA[1566,10] := 1.0;
   DATA[1566,11] := 19.74838;
   DATA[1566,12] := 2.212087;
   DATA[1566,13] := 914.0285;
   DATA[1566,14] := 1.0;
   DATA[1566,15] := 2.0;
   DATA[1566,16] := 1.0;
   DATA[1566,17] := 1.0;
   DATA[1566,18] := 1.0;
   DATA[1566,19] := 2.0;
   DATA[1566,20] := 148.808;
   DATA[1566,21] := 153.6785;
   DATA[1566,22] := 1.71262;
   DATA[1566,23] := 794.1041;
   DATA[1566,24] := 2.0;
   DATA[1566,25] := 2.0;
   DATA[1566,26] := 7.876378;
   DATA[1566,27] := 142.8608;
   DATA[1566,28] := 262.8172;
   DATA[1566,29] := 12.11228;
   DATA[1566,30] := 1.721866;
   DATA[1566,31] := 1.302293;
   DATA[1566,32] := 0.7352687;
   DATA[1566,33] := 0.3086827;
   DATA[1566,34] := 2.0;
   DATA[1566,35] := 249.984;
   DATA[1566,36] := 1.649953;
   DATA[1566,37] := 188.8138;
   DATA[1566,38] := 0.000128152;
   DATA[1566,39] := 1.0;
   DATA[1567,1] := 815.0835;
   DATA[1567,2] := 1.0;
   DATA[1567,3] := 1.0;
   DATA[1567,4] := 262.5288;
   DATA[1567,5] := 8.464369;
   DATA[1567,6] := 318.9695;
   DATA[1567,8] := 1.0;
   DATA[1567,9] := 1.0;
   DATA[1567,10] := 1.0;
   DATA[1567,11] := 19.71637;
   DATA[1567,12] := 2.212728;
   DATA[1567,13] := 913.7081;
   DATA[1567,14] := 1.0;
   DATA[1567,15] := 2.0;
   DATA[1567,16] := 1.0;
   DATA[1567,17] := 1.0;
   DATA[1567,18] := 1.0;
   DATA[1567,19] := 2.0;
   DATA[1567,20] := 148.808;
   DATA[1567,21] := 153.6785;
   DATA[1567,22] := 1.715567;
   DATA[1567,23] := 794.6039;
   DATA[1567,24] := 2.0;
   DATA[1567,25] := 2.0;
   DATA[1567,26] := 7.876378;
   DATA[1567,27] := 142.7839;
   DATA[1567,28] := 262.8172;
   DATA[1567,29] := 12.11228;
   DATA[1567,30] := 1.721866;
   DATA[1567,31] := 1.310106;
   DATA[1567,32] := 0.7352687;
   DATA[1567,33] := 0.3086827;
   DATA[1567,34] := 2.0;
   DATA[1567,35] := 249.984;
   DATA[1567,36] := 1.649953;
   DATA[1567,37] := 188.8138;
   DATA[1567,38] := 0.000128152;
   DATA[1567,39] := 1.0;
   DATA[1568,1] := 814.8873;
   DATA[1568,2] := 1.0;
   DATA[1568,3] := 1.0;
   DATA[1568,4] := 262.5288;
   DATA[1568,5] := 8.464369;
   DATA[1568,6] := 318.9695;
   DATA[1568,8] := 1.0;
   DATA[1568,9] := 1.0;
   DATA[1568,10] := 1.0;
   DATA[1568,11] := 19.69076;
   DATA[1568,12] := 2.214265;
   DATA[1568,13] := 912.8669;
   DATA[1568,14] := 1.0;
   DATA[1568,15] := 2.0;
   DATA[1568,16] := 1.0;
   DATA[1568,17] := 1.0;
   DATA[1568,18] := 1.0;
   DATA[1568,19] := 2.0;
   DATA[1568,20] := 148.808;
   DATA[1568,21] := 153.6785;
   DATA[1568,22] := 1.715567;
   DATA[1568,23] := 795.3345;
   DATA[1568,24] := 2.0;
   DATA[1568,25] := 2.0;
   DATA[1568,26] := 7.876378;
   DATA[1568,27] := 142.7839;
   DATA[1568,28] := 262.8172;
   DATA[1568,29] := 12.11228;
   DATA[1568,30] := 1.721866;
   DATA[1568,31] := 1.311643;
   DATA[1568,32] := 0.7352687;
   DATA[1568,33] := 0.3086827;
   DATA[1568,34] := 2.0;
   DATA[1568,35] := 249.984;
   DATA[1568,36] := 1.649953;
   DATA[1568,37] := 188.8138;
   DATA[1568,38] := 0.000128152;
   DATA[1568,39] := 1.0;
   DATA[1569,1] := 814.5732;
   DATA[1569,2] := 1.0;
   DATA[1569,3] := 1.0;
   DATA[1569,4] := 262.7211;
   DATA[1569,5] := 8.464369;
   DATA[1569,6] := 318.9695;
   DATA[1569,8] := 1.0;
   DATA[1569,9] := 1.0;
   DATA[1569,10] := 1.0;
   DATA[1569,11] := 19.69076;
   DATA[1569,12] := 2.214265;
   DATA[1569,13] := 912.7868;
   DATA[1569,14] := 1.0;
   DATA[1569,15] := 2.0;
   DATA[1569,16] := 1.0;
   DATA[1569,17] := 1.0;
   DATA[1569,18] := 1.0;
   DATA[1569,19] := 2.0;
   DATA[1569,20] := 148.808;
   DATA[1569,21] := 153.6785;
   DATA[1569,22] := 1.715567;
   DATA[1569,23] := 794.95;
   DATA[1569,24] := 2.0;
   DATA[1569,25] := 2.0;
   DATA[1569,26] := 7.876378;
   DATA[1569,27] := 142.7839;
   DATA[1569,28] := 262.8172;
   DATA[1569,29] := 12.11228;
   DATA[1569,30] := 1.724173;
   DATA[1569,31] := 1.312412;
   DATA[1569,32] := 0.7352687;
   DATA[1569,33] := 0.3082983;
   DATA[1569,34] := 2.0;
   DATA[1569,35] := 249.984;
   DATA[1569,36] := 1.649953;
   DATA[1569,37] := 188.8138;
   DATA[1569,38] := 0.000128152;
   DATA[1569,39] := 1.0;
   DATA[1570,1] := 814.2985;
   DATA[1570,2] := 1.0;
   DATA[1570,3] := 1.0;
   DATA[1570,4] := 262.7211;
   DATA[1570,5] := 8.464369;
   DATA[1570,6] := 318.9695;
   DATA[1570,8] := 1.0;
   DATA[1570,9] := 1.0;
   DATA[1570,10] := 1.0;
   DATA[1570,11] := 19.69076;
   DATA[1570,12] := 2.214265;
   DATA[1570,13] := 912.5865;
   DATA[1570,14] := 1.0;
   DATA[1570,15] := 2.0;
   DATA[1570,16] := 1.0;
   DATA[1570,17] := 1.0;
   DATA[1570,18] := 1.0;
   DATA[1570,19] := 2.0;
   DATA[1570,20] := 148.808;
   DATA[1570,21] := 153.6785;
   DATA[1570,22] := 1.715567;
   DATA[1570,23] := 795.1038;
   DATA[1570,24] := 2.0;
   DATA[1570,25] := 2.0;
   DATA[1570,26] := 7.876378;
   DATA[1570,27] := 142.7839;
   DATA[1570,28] := 262.8172;
   DATA[1570,29] := 12.11228;
   DATA[1570,30] := 1.724301;
   DATA[1570,31] := 1.308057;
   DATA[1570,32] := 0.7352687;
   DATA[1570,33] := 0.3081703;
   DATA[1570,34] := 2.0;
   DATA[1570,35] := 249.984;
   DATA[1570,36] := 1.649953;
   DATA[1570,37] := 188.8138;
   DATA[1570,38] := 0.000128152;
   DATA[1570,39] := 1.0;
   DATA[1571,1] := 814.2985;
   DATA[1571,2] := 1.0;
   DATA[1571,3] := 1.0;
   DATA[1571,4] := 262.7211;
   DATA[1571,5] := 8.464369;
   DATA[1571,6] := 318.9695;
   DATA[1571,8] := 1.0;
   DATA[1571,9] := 1.0;
   DATA[1571,10] := 1.0;
   DATA[1571,11] := 19.69076;
   DATA[1571,12] := 2.214265;
   DATA[1571,13] := 911.9857;
   DATA[1571,14] := 1.0;
   DATA[1571,15] := 2.0;
   DATA[1571,16] := 1.0;
   DATA[1571,17] := 1.0;
   DATA[1571,18] := 1.0;
   DATA[1571,19] := 2.0;
   DATA[1571,20] := 148.808;
   DATA[1571,21] := 153.6785;
   DATA[1571,22] := 1.712107;
   DATA[1571,23] := 795.3345;
   DATA[1571,24] := 2.0;
   DATA[1571,25] := 2.0;
   DATA[1571,26] := 7.876378;
   DATA[1571,27] := 142.7839;
   DATA[1571,28] := 262.8172;
   DATA[1571,29] := 12.11228;
   DATA[1571,30] := 1.724301;
   DATA[1571,31] := 1.29307;
   DATA[1571,32] := 0.7352687;
   DATA[1571,33] := 0.3081703;
   DATA[1571,34] := 2.0;
   DATA[1571,35] := 249.984;
   DATA[1571,36] := 1.649953;
   DATA[1571,37] := 188.8138;
   DATA[1571,38] := 0.000128152;
   DATA[1571,39] := 1.0;
   DATA[1572,1] := 814.4162;
   DATA[1572,2] := 1.0;
   DATA[1572,3] := 1.0;
   DATA[1572,4] := 262.7211;
   DATA[1572,5] := 8.464369;
   DATA[1572,6] := 318.9695;
   DATA[1572,8] := 1.0;
   DATA[1572,9] := 1.0;
   DATA[1572,10] := 1.0;
   DATA[1572,11] := 19.61393;
   DATA[1572,12] := 2.214265;
   DATA[1572,13] := 912.0659;
   DATA[1572,14] := 1.0;
   DATA[1572,15] := 2.0;
   DATA[1572,16] := 1.0;
   DATA[1572,17] := 1.0;
   DATA[1572,18] := 1.0;
   DATA[1572,19] := 2.0;
   DATA[1572,20] := 148.808;
   DATA[1572,21] := 153.6785;
   DATA[1572,22] := 1.710954;
   DATA[1572,23] := 795.2576;
   DATA[1572,24] := 2.0;
   DATA[1572,25] := 2.0;
   DATA[1572,26] := 7.876378;
   DATA[1572,27] := 142.7839;
   DATA[1572,28] := 262.8172;
   DATA[1572,29] := 12.11228;
   DATA[1572,30] := 1.724301;
   DATA[1572,31] := 1.292046;
   DATA[1572,32] := 0.7352687;
   DATA[1572,33] := 0.3081703;
   DATA[1572,34] := 2.0;
   DATA[1572,35] := 249.984;
   DATA[1572,36] := 1.649953;
   DATA[1572,37] := 188.8138;
   DATA[1572,38] := 0.000128152;
   DATA[1572,39] := 1.0;
   DATA[1573,1] := 814.22;
   DATA[1573,2] := 1.0;
   DATA[1573,3] := 1.0;
   DATA[1573,4] := 262.7211;
   DATA[1573,5] := 8.464369;
   DATA[1573,6] := 318.9695;
   DATA[1573,8] := 1.0;
   DATA[1573,9] := 1.0;
   DATA[1573,10] := 1.0;
   DATA[1573,11] := 19.61393;
   DATA[1573,12] := 2.214265;
   DATA[1573,13] := 911.425;
   DATA[1573,14] := 1.0;
   DATA[1573,15] := 2.0;
   DATA[1573,16] := 1.0;
   DATA[1573,17] := 1.0;
   DATA[1573,18] := 1.0;
   DATA[1573,19] := 2.0;
   DATA[1573,20] := 148.808;
   DATA[1573,21] := 153.6785;
   DATA[1573,22] := 1.710954;
   DATA[1573,23] := 795.1807;
   DATA[1573,24] := 2.0;
   DATA[1573,25] := 2.0;
   DATA[1573,26] := 7.876378;
   DATA[1573,27] := 142.7839;
   DATA[1573,28] := 262.8172;
   DATA[1573,29] := 12.11228;
   DATA[1573,30] := 1.724301;
   DATA[1573,31] := 1.284232;
   DATA[1573,32] := 0.7352687;
   DATA[1573,33] := 0.3082983;
   DATA[1573,34] := 2.0;
   DATA[1573,35] := 249.984;
   DATA[1573,36] := 1.649953;
   DATA[1573,37] := 188.8138;
   DATA[1573,38] := 0.000128152;
   DATA[1573,39] := 1.0;
   DATA[1574,1] := 814.3377;
   DATA[1574,2] := 1.0;
   DATA[1574,3] := 1.0;
   DATA[1574,4] := 262.7211;
   DATA[1574,5] := 8.464369;
   DATA[1574,6] := 318.9695;
   DATA[1574,8] := 1.0;
   DATA[1574,9] := 1.0;
   DATA[1574,10] := 1.0;
   DATA[1574,11] := 19.61393;
   DATA[1574,12] := 2.214265;
   DATA[1574,13] := 911.1046;
   DATA[1574,14] := 1.0;
   DATA[1574,15] := 2.0;
   DATA[1574,16] := 1.0;
   DATA[1574,17] := 1.0;
   DATA[1574,18] := 1.0;
   DATA[1574,19] := 2.0;
   DATA[1574,20] := 148.808;
   DATA[1574,21] := 153.6785;
   DATA[1574,22] := 1.710954;
   DATA[1574,23] := 795.4883;
   DATA[1574,24] := 2.0;
   DATA[1574,25] := 2.0;
   DATA[1574,26] := 7.876378;
   DATA[1574,27] := 142.7839;
   DATA[1574,28] := 262.8172;
   DATA[1574,29] := 12.11228;
   DATA[1574,30] := 1.723404;
   DATA[1574,31] := 1.280902;
   DATA[1574,32] := 0.7352687;
   DATA[1574,33] := 0.3086186;
   DATA[1574,34] := 2.0;
   DATA[1574,35] := 249.984;
   DATA[1574,36] := 1.585878;
   DATA[1574,37] := 188.8138;
   DATA[1574,38] := 0.000128152;
   DATA[1574,39] := 1.0;
   DATA[1575,1] := 813.9844;
   DATA[1575,2] := 1.0;
   DATA[1575,3] := 1.0;
   DATA[1575,4] := 262.4968;
   DATA[1575,5] := 8.464369;
   DATA[1575,6] := 318.9695;
   DATA[1575,8] := 1.0;
   DATA[1575,9] := 1.0;
   DATA[1575,10] := 1.0;
   DATA[1575,11] := 19.66195;
   DATA[1575,12] := 2.214265;
   DATA[1575,13] := 910.0632;
   DATA[1575,14] := 1.0;
   DATA[1575,15] := 2.0;
   DATA[1575,16] := 1.0;
   DATA[1575,17] := 1.0;
   DATA[1575,18] := 1.0;
   DATA[1575,19] := 2.0;
   DATA[1575,20] := 148.808;
   DATA[1575,21] := 153.6785;
   DATA[1575,22] := 1.710954;
   DATA[1575,23] := 795.1423;
   DATA[1575,24] := 2.0;
   DATA[1575,25] := 2.0;
   DATA[1575,26] := 7.876378;
   DATA[1575,27] := 142.7839;
   DATA[1575,28] := 262.8172;
   DATA[1575,29] := 12.11228;
   DATA[1575,30] := 1.721738;
   DATA[1575,31] := 1.280902;
   DATA[1575,32] := 0.7352687;
   DATA[1575,33] := 0.3086186;
   DATA[1575,34] := 2.0;
   DATA[1575,35] := 249.984;
   DATA[1575,36] := 1.585878;
   DATA[1575,37] := 188.8138;
   DATA[1575,38] := 0.000128152;
   DATA[1575,39] := 1.0;
   DATA[1576,1] := 813.7882;
   DATA[1576,2] := 1.0;
   DATA[1576,3] := 1.0;
   DATA[1576,4] := 262.4968;
   DATA[1576,5] := 8.464369;
   DATA[1576,6] := 318.9695;
   DATA[1576,8] := 1.0;
   DATA[1576,9] := 1.0;
   DATA[1576,10] := 1.0;
   DATA[1576,11] := 19.73558;
   DATA[1576,12] := 2.211318;
   DATA[1576,13] := 909.6226;
   DATA[1576,14] := 1.0;
   DATA[1576,15] := 2.0;
   DATA[1576,16] := 1.0;
   DATA[1576,17] := 1.0;
   DATA[1576,18] := 1.0;
   DATA[1576,19] := 2.0;
   DATA[1576,20] := 148.808;
   DATA[1576,21] := 153.858;
   DATA[1576,22] := 1.714542;
   DATA[1576,23] := 795.1038;
   DATA[1576,24] := 2.0;
   DATA[1576,25] := 2.0;
   DATA[1576,26] := 7.876378;
   DATA[1576,27] := 142.8608;
   DATA[1576,28] := 262.8172;
   DATA[1576,29] := 12.11228;
   DATA[1576,30] := 1.721738;
   DATA[1576,31] := 1.288331;
   DATA[1576,32] := 0.7366771;
   DATA[1576,33] := 0.3086186;
   DATA[1576,34] := 2.0;
   DATA[1576,35] := 249.984;
   DATA[1576,36] := 1.585878;
   DATA[1576,37] := 188.8138;
   DATA[1576,38] := 0.000128152;
   DATA[1576,39] := 1.0;
   DATA[1577,1] := 813.9452;
   DATA[1577,2] := 1.0;
   DATA[1577,3] := 1.0;
   DATA[1577,4] := 262.4968;
   DATA[1577,5] := 8.464369;
   DATA[1577,6] := 318.9695;
   DATA[1577,8] := 1.0;
   DATA[1577,9] := 1.0;
   DATA[1577,10] := 1.0;
   DATA[1577,11] := 19.73558;
   DATA[1577,12] := 2.211318;
   DATA[1577,13] := 909.2621;
   DATA[1577,14] := 1.0;
   DATA[1577,15] := 2.0;
   DATA[1577,16] := 1.0;
   DATA[1577,17] := 1.0;
   DATA[1577,18] := 1.0;
   DATA[1577,19] := 2.0;
   DATA[1577,20] := 148.808;
   DATA[1577,21] := 153.858;
   DATA[1577,22] := 1.714542;
   DATA[1577,23] := 794.9885;
   DATA[1577,24] := 2.0;
   DATA[1577,25] := 2.0;
   DATA[1577,26] := 7.876378;
   DATA[1577,27] := 142.8608;
   DATA[1577,28] := 262.8172;
   DATA[1577,29] := 12.11228;
   DATA[1577,30] := 1.721738;
   DATA[1577,31] := 1.286282;
   DATA[1577,32] := 0.7366771;
   DATA[1577,33] := 0.3086186;
   DATA[1577,34] := 2.0;
   DATA[1577,35] := 250.0641;
   DATA[1577,36] := 1.585878;
   DATA[1577,37] := 189.022;
   DATA[1577,38] := 0.000128152;
   DATA[1577,39] := 1.0;
   DATA[1578,1] := 814.1022;
   DATA[1578,2] := 1.0;
   DATA[1578,3] := 1.0;
   DATA[1578,4] := 262.4968;
   DATA[1578,5] := 8.464369;
   DATA[1578,6] := 319.3027;
   DATA[1578,8] := 1.0;
   DATA[1578,9] := 1.0;
   DATA[1578,10] := 1.0;
   DATA[1578,11] := 19.73558;
   DATA[1578,12] := 2.214265;
   DATA[1578,13] := 908.8215;
   DATA[1578,14] := 1.0;
   DATA[1578,15] := 2.0;
   DATA[1578,16] := 1.0;
   DATA[1578,17] := 1.0;
   DATA[1578,18] := 1.0;
   DATA[1578,19] := 2.0;
   DATA[1578,20] := 148.808;
   DATA[1578,21] := 153.858;
   DATA[1578,22] := 1.714542;
   DATA[1578,23] := 794.8731;
   DATA[1578,24] := 2.0;
   DATA[1578,25] := 2.0;
   DATA[1578,26] := 7.876378;
   DATA[1578,27] := 142.8608;
   DATA[1578,28] := 262.8172;
   DATA[1578,29] := 12.11228;
   DATA[1578,30] := 1.724173;
   DATA[1578,31] := 1.290765;
   DATA[1578,32] := 0.7366771;
   DATA[1578,33] := 0.3086186;
   DATA[1578,34] := 2.0;
   DATA[1578,35] := 250.3044;
   DATA[1578,36] := 1.665972;
   DATA[1578,37] := 189.1182;
   DATA[1578,38] := 0.000128152;
   DATA[1578,39] := 1.0;
   DATA[1579,1] := 813.9452;
   DATA[1579,2] := 1.0;
   DATA[1579,3] := 1.0;
   DATA[1579,4] := 262.4968;
   DATA[1579,5] := 8.464369;
   DATA[1579,6] := 319.3027;
   DATA[1579,8] := 1.0;
   DATA[1579,9] := 1.0;
   DATA[1579,10] := 1.0;
   DATA[1579,11] := 19.73558;
   DATA[1579,12] := 2.214265;
   DATA[1579,13] := 908.461;
   DATA[1579,14] := 1.0;
   DATA[1579,15] := 2.0;
   DATA[1579,16] := 1.0;
   DATA[1579,17] := 1.0;
   DATA[1579,18] := 1.0;
   DATA[1579,19] := 2.0;
   DATA[1579,20] := 148.808;
   DATA[1579,21] := 153.858;
   DATA[1579,22] := 1.714542;
   DATA[1579,23] := 794.8731;
   DATA[1579,24] := 2.0;
   DATA[1579,25] := 2.0;
   DATA[1579,26] := 7.876378;
   DATA[1579,27] := 142.8608;
   DATA[1579,28] := 262.8172;
   DATA[1579,29] := 12.11228;
   DATA[1579,30] := 1.724301;
   DATA[1579,31] := 1.291789;
   DATA[1579,32] := 0.7378293;
   DATA[1579,33] := 0.3084265;
   DATA[1579,34] := 2.0;
   DATA[1579,35] := 250.4166;
   DATA[1579,36] := 1.665972;
   DATA[1579,37] := 189.1182;
   DATA[1579,38] := 0.000128152;
   DATA[1579,39] := 1.0;
   DATA[1580,1] := 813.7489;
   DATA[1580,2] := 1.0;
   DATA[1580,3] := 1.0;
   DATA[1580,4] := 262.4968;
   DATA[1580,5] := 8.464369;
   DATA[1580,6] := 319.3027;
   DATA[1580,8] := 1.0;
   DATA[1580,9] := 1.0;
   DATA[1580,10] := 1.0;
   DATA[1580,11] := 19.71637;
   DATA[1580,12] := 2.214265;
   DATA[1580,13] := 908.0204;
   DATA[1580,14] := 1.0;
   DATA[1580,15] := 2.0;
   DATA[1580,16] := 1.0;
   DATA[1580,17] := 1.0;
   DATA[1580,18] := 1.0;
   DATA[1580,19] := 2.0;
   DATA[1580,20] := 148.808;
   DATA[1580,21] := 153.858;
   DATA[1580,22] := 1.713645;
   DATA[1580,23] := 795.0654;
   DATA[1580,24] := 2.0;
   DATA[1580,25] := 2.0;
   DATA[1580,26] := 7.876378;
   DATA[1580,27] := 142.8608;
   DATA[1580,28] := 262.8172;
   DATA[1580,29] := 12.11228;
   DATA[1580,30] := 1.724301;
   DATA[1580,31] := 1.291789;
   DATA[1580,32] := 0.7391096;
   DATA[1580,33] := 0.3081703;
   DATA[1580,34] := 2.0;
   DATA[1580,35] := 250.4166;
   DATA[1580,36] := 1.665972;
   DATA[1580,37] := 189.1182;
   DATA[1580,38] := 0.000128152;
   DATA[1580,39] := 1.0;
   DATA[1581,1] := 813.9059;
   DATA[1581,2] := 1.0;
   DATA[1581,3] := 1.0;
   DATA[1581,4] := 262.4968;
   DATA[1581,5] := 8.464369;
   DATA[1581,6] := 319.3027;
   DATA[1581,8] := 1.0;
   DATA[1581,9] := 1.0;
   DATA[1581,10] := 1.0;
   DATA[1581,11] := 19.70677;
   DATA[1581,12] := 2.214265;
   DATA[1581,13] := 907.7801;
   DATA[1581,14] := 1.0;
   DATA[1581,15] := 2.0;
   DATA[1581,16] := 1.0;
   DATA[1581,17] := 1.0;
   DATA[1581,18] := 1.0;
   DATA[1581,19] := 2.0;
   DATA[1581,20] := 148.808;
   DATA[1581,21] := 153.858;
   DATA[1581,22] := 1.713645;
   DATA[1581,23] := 795.2961;
   DATA[1581,24] := 2.0;
   DATA[1581,25] := 2.0;
   DATA[1581,26] := 7.876378;
   DATA[1581,27] := 142.8608;
   DATA[1581,28] := 262.8172;
   DATA[1581,29] := 12.11228;
   DATA[1581,30] := 1.725711;
   DATA[1581,31] := 1.291149;
   DATA[1581,32] := 0.736421;
   DATA[1581,33] := 0.3081703;
   DATA[1581,34] := 2.0;
   DATA[1581,35] := 250.4166;
   DATA[1581,36] := 1.665972;
   DATA[1581,37] := 189.2143;
   DATA[1581,38] := 0.000128152;
   DATA[1581,39] := 1.0;
   DATA[1582,1] := 813.7882;
   DATA[1582,2] := 1.0;
   DATA[1582,3] := 1.0;
   DATA[1582,4] := 262.4968;
   DATA[1582,5] := 8.464369;
   DATA[1582,6] := 319.2771;
   DATA[1582,8] := 1.0;
   DATA[1582,9] := 1.0;
   DATA[1582,10] := 1.0;
   DATA[1582,11] := 19.70677;
   DATA[1582,12] := 2.214265;
   DATA[1582,13] := 907.6199;
   DATA[1582,14] := 1.0;
   DATA[1582,15] := 2.0;
   DATA[1582,16] := 1.0;
   DATA[1582,17] := 1.0;
   DATA[1582,18] := 1.0;
   DATA[1582,19] := 2.0;
   DATA[1582,20] := 148.808;
   DATA[1582,21] := 153.858;
   DATA[1582,22] := 1.713645;
   DATA[1582,23] := 795.3345;
   DATA[1582,24] := 2.0;
   DATA[1582,25] := 2.0;
   DATA[1582,26] := 7.876378;
   DATA[1582,27] := 143.1684;
   DATA[1582,28] := 262.8172;
   DATA[1582,29] := 12.11228;
   DATA[1582,30] := 1.726609;
   DATA[1582,31] := 1.282439;
   DATA[1582,32] := 0.7346286;
   DATA[1582,33] := 0.306761;
   DATA[1582,34] := 2.0;
   DATA[1582,35] := 250.4166;
   DATA[1582,36] := 1.665972;
   DATA[1582,37] := 189.2143;
   DATA[1582,38] := 0.000128152;
   DATA[1582,39] := 1.0;
   DATA[1583,1] := 813.9059;
   DATA[1583,2] := 1.0;
   DATA[1583,3] := 1.0;
   DATA[1583,4] := 262.4968;
   DATA[1583,5] := 8.465651;
   DATA[1583,6] := 319.2258;
   DATA[1583,8] := 1.0;
   DATA[1583,9] := 1.0;
   DATA[1583,10] := 1.0;
   DATA[1583,11] := 19.70677;
   DATA[1583,12] := 2.214265;
   DATA[1583,13] := 906.8989;
   DATA[1583,14] := 1.0;
   DATA[1583,15] := 2.0;
   DATA[1583,16] := 1.0;
   DATA[1583,17] := 1.0;
   DATA[1583,18] := 1.0;
   DATA[1583,19] := 2.0;
   DATA[1583,20] := 148.808;
   DATA[1583,21] := 153.858;
   DATA[1583,22] := 1.715952;
   DATA[1583,23] := 795.7575;
   DATA[1583,24] := 2.0;
   DATA[1583,25] := 2.0;
   DATA[1583,26] := 7.876378;
   DATA[1583,27] := 143.1684;
   DATA[1583,28] := 262.8172;
   DATA[1583,29] := 12.11228;
   DATA[1583,30] := 1.726609;
   DATA[1583,31] := 1.269502;
   DATA[1583,32] := 0.7346286;
   DATA[1583,33] := 0.306761;
   DATA[1583,34] := 2.0;
   DATA[1583,35] := 250.4166;
   DATA[1583,36] := 1.665972;
   DATA[1583,37] := 189.2143;
   DATA[1583,38] := 0.000128152;
   DATA[1583,39] := 1.0;
   DATA[1584,1] := 813.6312;
   DATA[1584,2] := 1.0;
   DATA[1584,3] := 1.0;
   DATA[1584,4] := 262.4968;
   DATA[1584,5] := 8.465651;
   DATA[1584,6] := 319.072;
   DATA[1584,8] := 1.0;
   DATA[1584,9] := 1.0;
   DATA[1584,10] := 1.0;
   DATA[1584,11] := 19.67155;
   DATA[1584,12] := 2.214265;
   DATA[1584,13] := 906.4583;
   DATA[1584,14] := 1.0;
   DATA[1584,15] := 2.0;
   DATA[1584,16] := 1.0;
   DATA[1584,17] := 1.0;
   DATA[1584,18] := 1.0;
   DATA[1584,19] := 2.0;
   DATA[1584,20] := 148.808;
   DATA[1584,21] := 153.858;
   DATA[1584,22] := 1.715952;
   DATA[1584,23] := 795.6806;
   DATA[1584,24] := 2.0;
   DATA[1584,25] := 2.0;
   DATA[1584,26] := 7.876378;
   DATA[1584,27] := 143.1684;
   DATA[1584,28] := 262.8172;
   DATA[1584,29] := 12.11228;
   DATA[1584,30] := 1.726609;
   DATA[1584,31] := 1.261304;
   DATA[1584,32] := 0.7346286;
   DATA[1584,33] := 0.306761;
   DATA[1584,34] := 2.0;
   DATA[1584,35] := 250.4166;
   DATA[1584,36] := 1.665972;
   DATA[1584,37] := 189.2143;
   DATA[1584,38] := 0.000128152;
   DATA[1584,39] := 1.0;
   DATA[1585,1] := 813.5919;
   DATA[1585,2] := 1.0;
   DATA[1585,3] := 1.0;
   DATA[1585,4] := 262.6891;
   DATA[1585,5] := 8.465651;
   DATA[1585,6] := 319.072;
   DATA[1585,8] := 1.0;
   DATA[1585,9] := 1.0;
   DATA[1585,10] := 1.0;
   DATA[1585,11] := 19.67155;
   DATA[1585,12] := 2.214265;
   DATA[1585,13] := 905.6172;
   DATA[1585,14] := 1.0;
   DATA[1585,15] := 2.0;
   DATA[1585,16] := 1.0;
   DATA[1585,17] := 1.0;
   DATA[1585,18] := 1.0;
   DATA[1585,19] := 2.0;
   DATA[1585,20] := 148.808;
   DATA[1585,21] := 153.858;
   DATA[1585,22] := 1.713389;
   DATA[1585,23] := 795.796;
   DATA[1585,24] := 2.0;
   DATA[1585,25] := 2.0;
   DATA[1585,26] := 7.876378;
   DATA[1585,27] := 143.1684;
   DATA[1585,28] := 262.8172;
   DATA[1585,29] := 12.11228;
   DATA[1585,30] := 1.726609;
   DATA[1585,31] := 1.26361;
   DATA[1585,32] := 0.7346286;
   DATA[1585,33] := 0.3084265;
   DATA[1585,34] := 2.0;
   DATA[1585,35] := 250.4166;
   DATA[1585,36] := 1.665972;
   DATA[1585,37] := 189.2143;
   DATA[1585,38] := 0.000128152;
   DATA[1585,39] := 1.0;
   DATA[1586,1] := 813.3956;
   DATA[1586,2] := 1.0;
   DATA[1586,3] := 1.0;
   DATA[1586,4] := 262.6891;
   DATA[1586,5] := 8.465651;
   DATA[1586,6] := 319.072;
   DATA[1586,8] := 1.0;
   DATA[1586,9] := 1.0;
   DATA[1586,10] := 1.0;
   DATA[1586,11] := 19.67155;
   DATA[1586,12] := 2.212856;
   DATA[1586,13] := 905.7774;
   DATA[1586,14] := 1.0;
   DATA[1586,15] := 2.0;
   DATA[1586,16] := 1.0;
   DATA[1586,17] := 1.0;
   DATA[1586,18] := 1.0;
   DATA[1586,19] := 2.0;
   DATA[1586,20] := 148.808;
   DATA[1586,21] := 153.858;
   DATA[1586,22] := 1.713004;
   DATA[1586,23] := 795.796;
   DATA[1586,24] := 2.0;
   DATA[1586,25] := 2.0;
   DATA[1586,26] := 7.874776;
   DATA[1586,27] := 143.0659;
   DATA[1586,28] := 262.8172;
   DATA[1586,29] := 12.11228;
   DATA[1586,30] := 1.726865;
   DATA[1586,31] := 1.271039;
   DATA[1586,32] := 0.7357808;
   DATA[1586,33] := 0.3084265;
   DATA[1586,34] := 2.0;
   DATA[1586,35] := 250.4166;
   DATA[1586,36] := 1.665972;
   DATA[1586,37] := 189.2143;
   DATA[1586,38] := 0.000128152;
   DATA[1586,39] := 1.0;
   DATA[1587,1] := 814.0237;
   DATA[1587,2] := 1.0;
   DATA[1587,3] := 1.0;
   DATA[1587,4] := 262.6891;
   DATA[1587,5] := 8.465651;
   DATA[1587,6] := 319.072;
   DATA[1587,8] := 1.0;
   DATA[1587,9] := 1.0;
   DATA[1587,10] := 1.0;
   DATA[1587,11] := 19.71637;
   DATA[1587,12] := 2.2126;
   DATA[1587,13] := 904.9763;
   DATA[1587,14] := 1.0;
   DATA[1587,15] := 2.0;
   DATA[1587,16] := 1.0;
   DATA[1587,17] := 1.0;
   DATA[1587,18] := 1.0;
   DATA[1587,19] := 2.0;
   DATA[1587,20] := 148.808;
   DATA[1587,21] := 153.9862;
   DATA[1587,22] := 1.713004;
   DATA[1587,23] := 796.1036;
   DATA[1587,24] := 2.0;
   DATA[1587,25] := 2.0;
   DATA[1587,26] := 7.874776;
   DATA[1587,27] := 143.0659;
   DATA[1587,28] := 262.8172;
   DATA[1587,29] := 12.11228;
   DATA[1587,30] := 1.726865;
   DATA[1587,31] := 1.280902;
   DATA[1587,32] := 0.7357808;
   DATA[1587,33] := 0.3084265;
   DATA[1587,34] := 2.0;
   DATA[1587,35] := 250.4166;
   DATA[1587,36] := 1.665972;
   DATA[1587,37] := 189.2143;
   DATA[1587,38] := 0.000128152;
   DATA[1587,39] := 1.0;
   DATA[1588,1] := 813.9844;
   DATA[1588,2] := 1.0;
   DATA[1588,3] := 1.0;
   DATA[1588,4] := 262.6891;
   DATA[1588,5] := 8.465651;
   DATA[1588,6] := 319.072;
   DATA[1588,8] := 1.0;
   DATA[1588,9] := 1.0;
   DATA[1588,10] := 1.0;
   DATA[1588,11] := 19.71637;
   DATA[1588,12] := 2.2126;
   DATA[1588,13] := 904.4957;
   DATA[1588,14] := 1.0;
   DATA[1588,15] := 2.0;
   DATA[1588,16] := 1.0;
   DATA[1588,17] := 1.0;
   DATA[1588,18] := 1.0;
   DATA[1588,19] := 2.0;
   DATA[1588,20] := 148.808;
   DATA[1588,21] := 153.9862;
   DATA[1588,22] := 1.713004;
   DATA[1588,23] := 796.1805;
   DATA[1588,24] := 2.0;
   DATA[1588,25] := 2.0;
   DATA[1588,26] := 7.874776;
   DATA[1588,27] := 143.0659;
   DATA[1588,28] := 262.8172;
   DATA[1588,29] := 12.11228;
   DATA[1588,30] := 1.726865;
   DATA[1588,31] := 1.28167;
   DATA[1588,32] := 0.7357808;
   DATA[1588,33] := 0.3084265;
   DATA[1588,34] := 2.0;
   DATA[1588,35] := 250.4166;
   DATA[1588,36] := 1.665972;
   DATA[1588,37] := 189.2143;
   DATA[1588,38] := 0.000128152;
   DATA[1588,39] := 1.0;
   DATA[1589,1] := 813.7489;
   DATA[1589,2] := 1.0;
   DATA[1589,3] := 1.0;
   DATA[1589,4] := 262.6891;
   DATA[1589,5] := 8.465651;
   DATA[1589,6] := 319.072;
   DATA[1589,8] := 1.0;
   DATA[1589,9] := 1.0;
   DATA[1589,10] := 1.0;
   DATA[1589,11] := 19.74838;
   DATA[1589,12] := 2.2126;
   DATA[1589,13] := 903.8948;
   DATA[1589,14] := 1.0;
   DATA[1589,15] := 2.0;
   DATA[1589,16] := 1.0;
   DATA[1589,17] := 1.0;
   DATA[1589,18] := 1.0;
   DATA[1589,19] := 2.0;
   DATA[1589,20] := 148.808;
   DATA[1589,21] := 153.9862;
   DATA[1589,22] := 1.71262;
   DATA[1589,23] := 795.9498;
   DATA[1589,24] := 2.0;
   DATA[1589,25] := 2.0;
   DATA[1589,26] := 7.874776;
   DATA[1589,27] := 143.0659;
   DATA[1589,28] := 262.8172;
   DATA[1589,29] := 12.11228;
   DATA[1589,30] := 1.726865;
   DATA[1589,31] := 1.279877;
   DATA[1589,32] := 0.7357808;
   DATA[1589,33] := 0.3084265;
   DATA[1589,34] := 2.0;
   DATA[1589,35] := 250.4166;
   DATA[1589,36] := 1.665972;
   DATA[1589,37] := 189.2143;
   DATA[1589,38] := 0.000128152;
   DATA[1589,39] := 1.0;
   DATA[1590,1] := 813.7489;
   DATA[1590,2] := 1.0;
   DATA[1590,3] := 1.0;
   DATA[1590,4] := 262.6891;
   DATA[1590,5] := 8.465651;
   DATA[1590,6] := 319.072;
   DATA[1590,8] := 1.0;
   DATA[1590,9] := 1.0;
   DATA[1590,10] := 1.0;
   DATA[1590,11] := 19.77079;
   DATA[1590,12] := 2.2126;
   DATA[1590,13] := 903.2941;
   DATA[1590,14] := 1.0;
   DATA[1590,15] := 2.0;
   DATA[1590,16] := 1.0;
   DATA[1590,17] := 1.0;
   DATA[1590,18] := 1.0;
   DATA[1590,19] := 2.0;
   DATA[1590,20] := 148.808;
   DATA[1590,21] := 153.9862;
   DATA[1590,22] := 1.711595;
   DATA[1590,23] := 796.3727;
   DATA[1590,24] := 2.0;
   DATA[1590,25] := 2.0;
   DATA[1590,26] := 7.874776;
   DATA[1590,27] := 143.0403;
   DATA[1590,28] := 262.8172;
   DATA[1590,29] := 11.92002;
   DATA[1590,30] := 1.726865;
   DATA[1590,31] := 1.279237;
   DATA[1590,32] := 0.7357808;
   DATA[1590,33] := 0.3084265;
   DATA[1590,34] := 2.0;
   DATA[1590,35] := 250.4166;
   DATA[1590,36] := 1.665972;
   DATA[1590,37] := 189.2143;
   DATA[1590,38] := 0.000128152;
   DATA[1590,39] := 1.0;
   DATA[1591,1] := 813.8275;
   DATA[1591,2] := 1.0;
   DATA[1591,3] := 1.0;
   DATA[1591,4] := 262.6891;
   DATA[1591,5] := 8.465651;
   DATA[1591,6] := 319.072;
   DATA[1591,8] := 1.0;
   DATA[1591,9] := 1.0;
   DATA[1591,10] := 1.0;
   DATA[1591,11] := 19.7996;
   DATA[1591,12] := 2.2126;
   DATA[1591,13] := 902.6532;
   DATA[1591,14] := 1.0;
   DATA[1591,15] := 2.0;
   DATA[1591,16] := 1.0;
   DATA[1591,17] := 1.0;
   DATA[1591,18] := 1.0;
   DATA[1591,19] := 2.0;
   DATA[1591,20] := 148.808;
   DATA[1591,21] := 153.9862;
   DATA[1591,22] := 1.711082;
   DATA[1591,23] := 796.5266;
   DATA[1591,24] := 2.0;
   DATA[1591,25] := 2.0;
   DATA[1591,26] := 7.874776;
   DATA[1591,27] := 143.0403;
   DATA[1591,28] := 262.8172;
   DATA[1591,29] := 11.92002;
   DATA[1591,30] := 1.726865;
   DATA[1591,31] := 1.28167;
   DATA[1591,32] := 0.7352687;
   DATA[1591,33] := 0.3084265;
   DATA[1591,34] := 2.0;
   DATA[1591,35] := 250.4166;
   DATA[1591,36] := 1.665972;
   DATA[1591,37] := 189.2143;
   DATA[1591,38] := 0.000128152;
   DATA[1591,39] := 1.0;
   DATA[1592,1] := 813.5134;
   DATA[1592,2] := 1.0;
   DATA[1592,3] := 1.0;
   DATA[1592,4] := 262.6891;
   DATA[1592,5] := 8.465651;
   DATA[1592,6] := 319.072;
   DATA[1592,8] := 1.0;
   DATA[1592,9] := 1.0;
   DATA[1592,10] := 1.0;
   DATA[1592,11] := 19.7996;
   DATA[1592,12] := 2.211318;
   DATA[1592,13] := 902.2126;
   DATA[1592,14] := 1.0;
   DATA[1592,15] := 2.0;
   DATA[1592,16] := 1.0;
   DATA[1592,17] := 1.0;
   DATA[1592,18] := 1.0;
   DATA[1592,19] := 2.0;
   DATA[1592,20] := 148.808;
   DATA[1592,21] := 153.9862;
   DATA[1592,22] := 1.7098;
   DATA[1592,23] := 796.4496;
   DATA[1592,24] := 2.0;
   DATA[1592,25] := 2.0;
   DATA[1592,26] := 7.874776;
   DATA[1592,27] := 143.0403;
   DATA[1592,28] := 262.8172;
   DATA[1592,29] := 11.92002;
   DATA[1592,30] := 1.726865;
   DATA[1592,31] := 1.291405;
   DATA[1592,32] := 0.7351407;
   DATA[1592,33] := 0.3084265;
   DATA[1592,34] := 2.0;
   DATA[1592,35] := 250.4166;
   DATA[1592,36] := 1.665972;
   DATA[1592,37] := 189.2143;
   DATA[1592,38] := 0.000128152;
   DATA[1592,39] := 1.0;
   DATA[1593,1] := 813.7489;
   DATA[1593,2] := 1.0;
   DATA[1593,3] := 1.0;
   DATA[1593,4] := 262.6891;
   DATA[1593,5] := 8.465651;
   DATA[1593,6] := 319.072;
   DATA[1593,8] := 1.0;
   DATA[1593,9] := 1.0;
   DATA[1593,10] := 1.0;
   DATA[1593,11] := 19.73878;
   DATA[1593,12] := 2.211318;
   DATA[1593,13] := 901.772;
   DATA[1593,14] := 1.0;
   DATA[1593,15] := 2.0;
   DATA[1593,16] := 1.0;
   DATA[1593,17] := 1.0;
   DATA[1593,18] := 1.0;
   DATA[1593,19] := 2.0;
   DATA[1593,20] := 148.808;
   DATA[1593,21] := 153.9862;
   DATA[1593,22] := 1.7098;
   DATA[1593,23] := 796.565;
   DATA[1593,24] := 2.0;
   DATA[1593,25] := 2.0;
   DATA[1593,26] := 7.874776;
   DATA[1593,27] := 143.0403;
   DATA[1593,28] := 262.8172;
   DATA[1593,29] := 11.92002;
   DATA[1593,30] := 1.726865;
   DATA[1593,31] := 1.285641;
   DATA[1593,32] := 0.7351407;
   DATA[1593,33] := 0.3084265;
   DATA[1593,34] := 2.0;
   DATA[1593,35] := 250.4166;
   DATA[1593,36] := 1.665972;
   DATA[1593,37] := 189.2143;
   DATA[1593,38] := 0.000128152;
   DATA[1593,39] := 1.0;
   DATA[1594,1] := 813.5919;
   DATA[1594,2] := 1.0;
   DATA[1594,3] := 1.0;
   DATA[1594,4] := 262.6891;
   DATA[1594,5] := 8.465651;
   DATA[1594,6] := 319.072;
   DATA[1594,8] := 1.0;
   DATA[1594,9] := 1.0;
   DATA[1594,10] := 1.0;
   DATA[1594,11] := 19.73878;
   DATA[1594,12] := 2.2126;
   DATA[1594,13] := 901.2914;
   DATA[1594,14] := 1.0;
   DATA[1594,15] := 2.0;
   DATA[1594,16] := 1.0;
   DATA[1594,17] := 1.0;
   DATA[1594,18] := 1.0;
   DATA[1594,19] := 2.0;
   DATA[1594,20] := 148.808;
   DATA[1594,21] := 153.9862;
   DATA[1594,22] := 1.7098;
   DATA[1594,23] := 797.1418;
   DATA[1594,24] := 2.0;
   DATA[1594,25] := 2.0;
   DATA[1594,26] := 7.874776;
   DATA[1594,27] := 142.8352;
   DATA[1594,28] := 262.8172;
   DATA[1594,29] := 11.92002;
   DATA[1594,30] := 1.726865;
   DATA[1594,31] := 1.289228;
   DATA[1594,32] := 0.7351407;
   DATA[1594,33] := 0.3084265;
   DATA[1594,34] := 2.0;
   DATA[1594,35] := 250.3044;
   DATA[1594,36] := 1.665972;
   DATA[1594,37] := 189.2143;
   DATA[1594,38] := 0.000128152;
   DATA[1594,39] := 1.0;
   DATA[1595,1] := 813.7882;
   DATA[1595,2] := 1.0;
   DATA[1595,3] := 1.0;
   DATA[1595,4] := 262.6891;
   DATA[1595,5] := 8.465651;
   DATA[1595,6] := 319.072;
   DATA[1595,8] := 1.0;
   DATA[1595,9] := 1.0;
   DATA[1595,10] := 1.0;
   DATA[1595,11] := 19.73878;
   DATA[1595,12] := 2.212856;
   DATA[1595,13] := 900.6906;
   DATA[1595,14] := 1.0;
   DATA[1595,15] := 2.0;
   DATA[1595,16] := 1.0;
   DATA[1595,17] := 1.0;
   DATA[1595,18] := 1.0;
   DATA[1595,19] := 2.0;
   DATA[1595,20] := 148.808;
   DATA[1595,21] := 153.9862;
   DATA[1595,22] := 1.7098;
   DATA[1595,23] := 797.0649;
   DATA[1595,24] := 2.0;
   DATA[1595,25] := 2.0;
   DATA[1595,26] := 7.877339;
   DATA[1595,27] := 142.8352;
   DATA[1595,28] := 262.8172;
   DATA[1595,29] := 11.92002;
   DATA[1595,30] := 1.726865;
   DATA[1595,31] := 1.291789;
   DATA[1595,32] := 0.7351407;
   DATA[1595,33] := 0.3084265;
   DATA[1595,34] := 2.0;
   DATA[1595,35] := 250.2724;
   DATA[1595,36] := 1.665972;
   DATA[1595,37] := 188.8939;
   DATA[1595,38] := 0.000128152;
   DATA[1595,39] := 1.0;
   DATA[1596,1] := 813.7882;
   DATA[1596,2] := 1.0;
   DATA[1596,3] := 1.0;
   DATA[1596,4] := 262.6891;
   DATA[1596,5] := 8.465651;
   DATA[1596,6] := 319.072;
   DATA[1596,8] := 1.0;
   DATA[1596,9] := 1.0;
   DATA[1596,10] := 1.0;
   DATA[1596,11] := 19.73878;
   DATA[1596,12] := 2.212856;
   DATA[1596,13] := 900.2499;
   DATA[1596,14] := 1.0;
   DATA[1596,15] := 2.0;
   DATA[1596,16] := 1.0;
   DATA[1596,17] := 1.0;
   DATA[1596,18] := 1.0;
   DATA[1596,19] := 2.0;
   DATA[1596,20] := 148.808;
   DATA[1596,21] := 153.9862;
   DATA[1596,22] := 1.7098;
   DATA[1596,23] := 797.2187;
   DATA[1596,24] := 2.0;
   DATA[1596,25] := 2.0;
   DATA[1596,26] := 7.877339;
   DATA[1596,27] := 142.8352;
   DATA[1596,28] := 262.8172;
   DATA[1596,29] := 12.26609;
   DATA[1596,30] := 1.725968;
   DATA[1596,31] := 1.291789;
   DATA[1596,32] := 0.7351407;
   DATA[1596,33] := 0.3084265;
   DATA[1596,34] := 2.0;
   DATA[1596,35] := 250.0801;
   DATA[1596,36] := 1.665972;
   DATA[1596,37] := 188.8779;
   DATA[1596,38] := 0.000128152;
   DATA[1596,39] := 1.0;
   DATA[1597,1] := 813.6312;
   DATA[1597,2] := 1.0;
   DATA[1597,3] := 1.0;
   DATA[1597,4] := 262.4648;
   DATA[1597,5] := 8.465651;
   DATA[1597,6] := 319.072;
   DATA[1597,8] := 1.0;
   DATA[1597,9] := 1.0;
   DATA[1597,10] := 1.0;
   DATA[1597,11] := 19.75159;
   DATA[1597,12] := 2.212856;
   DATA[1597,13] := 899.7693;
   DATA[1597,14] := 1.0;
   DATA[1597,15] := 2.0;
   DATA[1597,16] := 1.0;
   DATA[1597,17] := 1.0;
   DATA[1597,18] := 1.0;
   DATA[1597,19] := 2.0;
   DATA[1597,20] := 148.808;
   DATA[1597,21] := 153.9862;
   DATA[1597,22] := 1.7098;
   DATA[1597,23] := 797.4494;
   DATA[1597,24] := 2.0;
   DATA[1597,25] := 2.0;
   DATA[1597,26] := 7.877339;
   DATA[1597,27] := 142.8352;
   DATA[1597,28] := 262.8172;
   DATA[1597,29] := 12.26609;
   DATA[1597,30] := 1.724301;
   DATA[1597,31] := 1.301652;
   DATA[1597,32] := 0.7351407;
   DATA[1597,33] := 0.3084265;
   DATA[1597,34] := 2.0;
   DATA[1597,35] := 250.0801;
   DATA[1597,36] := 1.665972;
   DATA[1597,37] := 188.8779;
   DATA[1597,38] := 0.000128152;
   DATA[1597,39] := 1.0;
   DATA[1598,1] := 813.5134;
   DATA[1598,2] := 1.0;
   DATA[1598,3] := 1.0;
   DATA[1598,4] := 262.4648;
   DATA[1598,5] := 8.466612;
   DATA[1598,6] := 319.072;
   DATA[1598,8] := 1.0;
   DATA[1598,9] := 1.0;
   DATA[1598,10] := 1.0;
   DATA[1598,11] := 19.7804;
   DATA[1598,12] := 2.212856;
   DATA[1598,13] := 899.4489;
   DATA[1598,14] := 1.0;
   DATA[1598,15] := 2.0;
   DATA[1598,16] := 1.0;
   DATA[1598,17] := 1.0;
   DATA[1598,18] := 1.0;
   DATA[1598,19] := 2.0;
   DATA[1598,20] := 148.808;
   DATA[1598,21] := 153.9862;
   DATA[1598,22] := 1.7098;
   DATA[1598,23] := 797.5262;
   DATA[1598,24] := 2.0;
   DATA[1598,25] := 2.0;
   DATA[1598,26] := 7.877339;
   DATA[1598,27] := 143.0403;
   DATA[1598,28] := 262.8172;
   DATA[1598,29] := 12.26609;
   DATA[1598,30] := 1.722379;
   DATA[1598,31] := 1.294095;
   DATA[1598,32] := 0.7351407;
   DATA[1598,33] := 0.3074656;
   DATA[1598,34] := 2.0;
   DATA[1598,35] := 249.9359;
   DATA[1598,36] := 1.665972;
   DATA[1598,37] := 188.8779;
   DATA[1598,38] := 0.000128152;
   DATA[1598,39] := 1.0;
   DATA[1599,1] := 813.9059;
   DATA[1599,2] := 1.0;
   DATA[1599,3] := 1.0;
   DATA[1599,4] := 262.4648;
   DATA[1599,5] := 8.467573;
   DATA[1599,6] := 319.072;
   DATA[1599,8] := 1.0;
   DATA[1599,9] := 1.0;
   DATA[1599,10] := 1.0;
   DATA[1599,11] := 19.7964;
   DATA[1599,12] := 2.212856;
   DATA[1599,13] := 898.9282;
   DATA[1599,14] := 1.0;
   DATA[1599,15] := 2.0;
   DATA[1599,16] := 1.0;
   DATA[1599,17] := 1.0;
   DATA[1599,18] := 1.0;
   DATA[1599,19] := 2.0;
   DATA[1599,20] := 148.808;
   DATA[1599,21] := 153.9093;
   DATA[1599,22] := 1.7098;
   DATA[1599,23] := 797.4879;
   DATA[1599,24] := 2.0;
   DATA[1599,25] := 2.0;
   DATA[1599,26] := 7.877339;
   DATA[1599,27] := 143.0403;
   DATA[1599,28] := 262.8172;
   DATA[1599,29] := 12.26609;
   DATA[1599,30] := 1.722379;
   DATA[1599,31] := 1.291533;
   DATA[1599,32] := 0.7351407;
   DATA[1599,33] := 0.3074656;
   DATA[1599,34] := 2.0;
   DATA[1599,35] := 249.9359;
   DATA[1599,36] := 1.665972;
   DATA[1599,37] := 188.8779;
   DATA[1599,38] := 0.000128152;
   DATA[1599,39] := 1.0;
   DATA[1600,1] := 814.2985;
   DATA[1600,2] := 1.0;
   DATA[1600,3] := 1.0;
   DATA[1600,4] := 262.4648;
   DATA[1600,5] := 8.467573;
   DATA[1600,6] := 319.072;
   DATA[1600,8] := 1.0;
   DATA[1600,9] := 1.0;
   DATA[1600,10] := 1.0;
   DATA[1600,11] := 19.7964;
   DATA[1600,12] := 2.212856;
   DATA[1600,13] := 898.8481;
   DATA[1600,14] := 1.0;
   DATA[1600,15] := 2.0;
   DATA[1600,16] := 1.0;
   DATA[1600,17] := 1.0;
   DATA[1600,18] := 1.0;
   DATA[1600,19] := 2.0;
   DATA[1600,20] := 148.808;
   DATA[1600,21] := 153.858;
   DATA[1600,22] := 1.7098;
   DATA[1600,23] := 797.6416;
   DATA[1600,24] := 2.0;
   DATA[1600,25] := 2.0;
   DATA[1600,26] := 7.877339;
   DATA[1600,27] := 143.0403;
   DATA[1600,28] := 262.8172;
   DATA[1600,29] := 12.07383;
   DATA[1600,30] := 1.720969;
   DATA[1600,31] := 1.291533;
   DATA[1600,32] := 0.7351407;
